(* Logix 5000 project; controller VET 1756-L62 rev 19.52; software revision 19.01; part 6 of 27 *)

        [445].S.BITS2.27   // 9-CON-707 Cmd. Open
        [445].S.BITS2.30   // 9-CON-707 OUT CLOSE
        [445].S.BITS2.31   // 9-CON-707 OUT OPEN
        [447].S.BITS2.31   // 9-CON-709 OUT OPEN
        [450].S.BITS2.31   // 110-VEN-001/2 OUT MARCHA
        [451].S.BITS2.31   // 9-CON-713 OUT OPEN
        [462].S.BITS2.31   // 110-ENF-002/2-4 OUT MARCHA
        [464].S.BITS2.31   // 110-ENF-002/2-1 OUT MARCHA
        [465].S.BITS1.1   // 9-CON-727 Falla Resumen
        [465].S.BITS1.2   // 9-CON-727 Conf Pos Abrir
        [465].S.BITS1.4   // 9-CON-727 Conf Pos Cerrar
        [465].S.BITS1.29   // 9-CON-727 Falla Abrir
        [465].S.BITS1.30   // 9-CON-727 Falla Cerrar
        [465].S.BITS2.20   // 9-CON-727 Reset Falla
        [465].S.BITS2.27   // 9-CON-727 Cmd. Open
        [465].S.BITS2.30   // 9-CON-727 OUT CLOSE
        [465].S.BITS2.31   // 9-CON-727 OUT OPEN
        [467].S.BITS2.31   // 9-CON-729 OUT OPEN
        [471].S.BITS2.31   // 110-ENF-002/2-5 OUT MARCHA
        [474].S.BITS2.31   // 110-TOR-002/2 OUT MARCHA
        [475].S.BITS2.31   // 110-TOR-003/2 OUT MARCHA
        [476].S.BITS2.31   // 110-ELV-002/2 OUT MARCHA
        [478].S.BITS2.31   // 110-TOR-004/2 OUT MARCHA
        [495].S.BITS2.31   // 110-CAN-010/3 OUT MARCHA
        [500].S.BITS2.31   // 110-TOR-001/3 OUT MARCHA
        [502].S.BITS2.31   // 110-ACD-001/3 OUT MARCHA
        [504].S.BITS2.31   // 110-DES-001/3 OUT MARCHA
        [505].S.BITS2.31   // 110-CAE-001/3 OUT MARCHA
        [511].S.BITS2.31   // 110-ESC-001/3 OUT MARCHA
        [512].S.BITS2.31   // 110-ENF-001/3-4 OUT MARCHA
        [514].S.BITS2.31   // 110-ENF-001/3-1 OUT MARCHA
        [515].S.BITS1.1   // 110-ENF-001/3-2 Falla Resumen
        [515].S.BITS1.2   // 110-ENF-001/3-2 Conf Pos Abrir
        [515].S.BITS1.4   // 110-ENF-001/3-2 Conf Pos Cerrar
        [515].S.BITS1.29   // 110-ENF-001/3-2 Falla Abrir
        [515].S.BITS1.30   // 110-ENF-001/3-2 Falla Cerrar
        [515].S.BITS2.20   // 110-ENF-001/3-2 Reset Falla
        [515].S.BITS2.27   // 110-ENF-001/3-2 Cmd. Open
        [515].S.BITS2.30   // 110-ENF-001/3-2 OUT CLOSE
        [515].S.BITS2.31   // 110-ENF-001/3-2 OUT OPEN
        [517].S.BITS2.31   // 110-ESC-003/3 OUT MARCHA
        [519].S.BITS2.31   // 110-VAL-001/3-1 OUT MARCHA
        [520].S.BITS2.31   // 110-VEN-001/3 OUT MARCHA
        [521].S.BITS2.31   // 110-ENF-001/3-5 OUT MARCHA
        [523].S.BITS2.31   // 110-QUE-001-1 OUT MARCHA
        [524].S.BITS2.31   // 110-QUE-001-2 OUT MARCHA
        [531].S.BITS2.31   // 110-ESC-002/3 OUT MARCHA
        [532].S.BITS2.31   // 110-ENF-002/3-4 OUT MARCHA
        [534].S.BITS2.31   // 110-ENF-002/3-1 OUT MARCHA
        [535].S.BITS1.1   // 110-ENF-002/3-2 Falla Resumen
        [535].S.BITS1.2   // 110-ENF-002/3-2 Conf Pos Abrir
        [535].S.BITS1.4   // 110-ENF-002/3-2 Conf Pos Cerrar
        [535].S.BITS1.29   // 110-ENF-002/3-2 Falla Abrir
        [535].S.BITS1.30   // 110-ENF-002/3-2 Falla Cerrar
        [535].S.BITS2.20   // 110-ENF-002/3-2 Reset Falla
        [535].S.BITS2.27   // 110-ENF-002/3-2 Cmd. Open
        [535].S.BITS2.30   // 110-ENF-002/3-2 OUT CLOSE
        [535].S.BITS2.31   // 110-ENF-002/3-2 OUT OPEN
        [537].S.BITS2.31   // 110-ESC-004/3 OUT MARCHA
        [539].S.BITS2.31   // 110-VEN-002/3-1 OUT MARCHA
        [540].S.BITS2.31   // 110-VEN-002/3 OUT MARCHA
        [541].S.BITS2.31   // 110-ENF-002/3-5 OUT MARCHA
        [544].S.BITS2.31   // 110-TOR-002/3 OUT MARCHA
        [545].S.BITS2.31   // 110-TOR-003/3 OUT MARCHA
        [546].S.BITS2.31   // 110-ELV-002/3 OUT MARCHA
        [548].S.BITS2.31   // 110-TOR-004/3 OUT MARCHA
        [551].S.BITS2.31   // 110-TDC-003/1 OUT MARCHA
        [555].S.BITS2.31   // 120-TDC-001/1 OUT MARCHA
        [561].S.BITS2.31   // 110-TDC-003/2 OUT MARCHA
        [562].S.BITS2.31   // 110-TDC-004/2 OUT MARCHA
        [564].S.BITS2.31   // 110-ELV-001/2 OUT MARCHA
        [565].S.BITS2.31   // 120-TDC-001/2 OUT MARCHA
        [571].S.BITS2.31   // 110-TDC-003/3 OUT MARCHA
        [572].S.BITS2.31   // 110-TDC-004/3 OUT MARCHA
        [573].S.BITS2.31   // 110-TDC-005/3 OUT MARCHA
        [574].S.BITS2.31   // 110-ELV-001/3 OUT MARCHA
        [575].S.BITS2.31   // 120-TDC-001/3 OUT MARCHA
        [349].S.BITS1.7   // 110-LRT-001 Puerta
        [383].S.BITS1.14   // Switch de Incendio
        [383].S.BITS1.3   // Alineamiento plataforma
        [383].S.BITS1.11   // Puerta Abierta
        [691].S.BITS1.2   // 100-DOS-100-M13 Conf. Marcha
        [693].S.BITS1.2   // 100-DOS-100-M14 Conf. Marcha
        [1].S.BITS1.4   // 7-LMG-1001 Cmd. Automatico
        [1].S.BITS1.26   // 7-LMG-1001 FLL
        [1].S.BITS1.27   // 7-LMG-1001 FV0
        [1].S.BITS1.28   // 7-LMG-1001 FATO
        [1].S.BITS1.30   // 7-LMG-1001 Falla Partida
        [1].S.BITS2.27   // 7-LMG-1001 Cmd. Marcha
        [1].S.BITS2.20   // 7-LMG-1001 Reset Falla
        [1].S.BITS2.23   // 7-LMG-1001 Test
        [1].S.BITS2.30   // 7-LMG-1001 OUT MARCHA
        [2].S.BITS1.0   // 7-ELV-1002 Enable
        [2].S.BITS1.1   // 7-ELV-1002 Falla Resumen
        [2].S.BITS1.2   // 7-ELV-1002 Conf. Marcha
        [2].S.BITS1.4   // 7-ELV-1002 Cmd. Automatico
        [2].S.BITS1.26   // 7-ELV-1002 FLL
        [2].S.BITS1.27   // 7-ELV-1002 FV0
        [2].S.BITS1.28   // 7-ELV-1002 FATO
        [2].S.BITS1.30   // 7-ELV-1002 Falla Partida
        [2].S.BITS2.27   // 7-ELV-1002 Cmd. Marcha
        [2].S.BITS2.20   // 7-ELV-1002 Reset Falla
        [2].S.BITS2.23   // 7-ELV-1002 Test
        [2].S.BITS2.30   // 7-ELV-1002 OUT MARCHA
        [3].S.BITS1.0   // 7-BIF-1003 Enable
        [3].S.BITS1.1   // 7-BIF-1003 Falla Resumen
        [3].S.BITS1.2   // 7-BIF-1003 Conf. Pos. Izquierda
        [3].S.BITS1.4   // 7-BIF-1003 Conf. Pos. Derecha
        [3].S.BITS1.29   // 7-BIF-1003 Falla Pos. Izquierda
        [3].S.BITS1.30   // 7-BIF-1003 Falla Pos. Derecha
        [3].S.BITS2.20   // 7-BIF-1003 Reset Falla
        [3].S.BITS2.23   // 7-BIF-1003 Test
        [3].S.BITS2.26   // 7-BIF-1003 Cmd. Pos . Izquierda
        [3].S.BITS2.27   // 7-BIF-1003 Cmd. Pos. Derecha
        [3].S.BITS2.30   // 7-BIF-1003 Out Izquierda
        [3].S.BITS2.31   // 7-BIF-1003 Out Derecha
        [5].S.BITS1.26   // 7-RED-1005 FLL
        [5].S.BITS1.27   // 7-RED-1005 FV0
        [5].S.BITS1.28   // 7-RED-1005 FATO
        [5].S.BITS1.30   // 7-RED-1005 Falla Partida
        [5].S.BITS2.27   // 7-RED-1005 Cmd. Marcha
        [5].S.BITS2.30   // 7-RED-1005 OUT MARCHA
        [6].S.BITS2.31   // 7-COM-1006 OUT OPEN
        [8].S.BITS2.31   // 7-COM-1008 OUT OPEN
        [10].S.BITS1.0   // 7-RED-1010 Enable
        [10].S.BITS1.1   // 7-RED-1010 Falla Resumen
        [10].S.BITS1.2   // 7-RED-1010 Conf. Marcha
        [10].S.BITS1.4   // 7-RED-1010 Cmd. Automatico
        [10].S.BITS1.26   // 7-RED-1010 FLL
        [10].S.BITS1.27   // 7-RED-1010 FV0
        [10].S.BITS1.28   // 7-RED-1010 FATO
        [10].S.BITS1.30   // 7-RED-1010 Falla Partida
        [10].S.BITS2.27   // 7-RED-1010 Cmd. Marcha
        [10].S.BITS2.20   // 7-RED-1010 Reset Falla
        [10].S.BITS2.23   // 7-RED-1010 Test
        [10].S.BITS2.30   // 7-RED-1010 OUT MARCHA
        [11].S.BITS1.0   // 7-CON-1011 Enable
        [11].S.BITS1.1   // 7-CON-1011 Falla Resumen
        [11].S.BITS1.2   // 7-CON-1011 Conf Pos Abrir
        [11].S.BITS1.4   // 7-CON-1011 Conf Pos Cerrar
        [11].S.BITS1.29   // 7-CON-1011 Falla Abrir
        [11].S.BITS1.30   // 7-CON-1011 Falla Cerrar
        [11].S.BITS2.20   // 7-CON-1011 Reset Falla
        [11].S.BITS2.23   // 7-CON-1011 Test
        [11].S.BITS2.27   // 7-CON-1011 Cmd. Open
        [11].S.BITS2.30   // 7-CON-1011 OUT CLOSE
        [11].S.BITS2.31   // 7-CON-1011 OUT OPEN
        [12].S.BITS1.0   // 7-CON-1012 Enable
        [12].S.BITS1.1   // 7-CON-1012 Falla Resumen
        [12].S.BITS1.2   // 7-CON-1012 Conf Pos Abrir
        [12].S.BITS1.4   // 7-CON-1012 Conf Pos Cerrar
        [12].S.BITS1.29   // 7-CON-1012 Falla Abrir
        [12].S.BITS1.30   // 7-CON-1012 Falla Cerrar
        [12].S.BITS2.20   // 7-CON-1012 Reset Falla
        [12].S.BITS2.23   // 7-CON-1012 Test
        [12].S.BITS2.27   // 7-CON-1012 Cmd. Open
        [12].S.BITS2.30   // 7-CON-1012 OUT CLOSE
        [12].S.BITS2.31   // 7-CON-1012 OUT OPEN
        [13].S.BITS1.2   // 7-CON-1013 Conf Pos Abrir
        [15].S.BITS1.0   // 7-BIF-1023a Enable
        [15].S.BITS1.1   // 7-BIF-1023a Falla Resumen
        [15].S.BITS1.2   // 7-BIF-1023a Conf. Pos. Izquierda
        [15].S.BITS1.4   // 7-BIF-1023a Conf. Pos. Derecha
        [15].S.BITS1.29   // 7-BIF-1023a Falla Pos. Izquierda
        [15].S.BITS1.30   // 7-BIF-1023a Falla Pos. Derecha
        [15].S.BITS2.20   // 7-BIF-1023a Reset Falla
        [15].S.BITS2.23   // 7-BIF-1023a Test
        [15].S.BITS2.26   // 7-BIF-1023a Cmd. Pos . Izquierda
        [15].S.BITS2.27   // 7-BIF-1023a Cmd. Pos. Derecha
        [15].S.BITS2.30   // 7-BIF-1023a Out Izquierda
        [15].S.BITS2.31   // 7-BIF-1023a Out Derecha
        [16].S.BITS1.26   // 7-LMG-1016 FLL
        [16].S.BITS1.27   // 7-LMG-1016 FV0
        [16].S.BITS1.28   // 7-LMG-1016 FATO
        [16].S.BITS1.30   // 7-LMG-1016 Falla Partida
        [16].S.BITS2.27   // 7-LMG-1016 Cmd. Marcha
        [16].S.BITS2.30   // 7-LMG-1016 OUT MARCHA
        [17].S.BITS1.26   // 7-ELV-1017 FLL
        [17].S.BITS1.27   // 7-ELV-1017 FV0
        [17].S.BITS1.28   // 7-ELV-1017 FATO
        [17].S.BITS1.30   // 7-ELV-1017 Falla Partida
        [17].S.BITS2.27   // 7-ELV-1017 Cmd. Marcha
        [17].S.BITS2.30   // 7-ELV-1017 OUT MARCHA
        [18].S.BITS1.2   // 7-BIF-1018 Conf. Pos. Izquierda
        [18].S.BITS1.4   // 7-BIF-1018 Conf. Pos. Derecha
        [18].S.BITS1.29   // 7-BIF-1018 Falla Pos. Izquierda
        [18].S.BITS1.30   // 7-BIF-1018 Falla Pos. Derecha
        [18].S.BITS2.26   // 7-BIF-1018 Cmd. Pos . Izquierda
        [18].S.BITS2.27   // 7-BIF-1018 Cmd. Pos. Derecha
        [18].S.BITS2.30   // 7-BIF-1018 Out Izquierda
        [18].S.BITS2.31   // 7-BIF-1018 Out Derecha
        [19].S.BITS1.26   // 7-RED-1019 FLL
        [19].S.BITS1.27   // 7-RED-1019 FV0
        [19].S.BITS1.28   // 7-RED-1019 FATO
        [19].S.BITS1.30   // 7-RED-1019 Falla Partida
        [19].S.BITS2.27   // 7-RED-1019 Cmd. Marcha
        [19].S.BITS2.30   // 7-RED-1019 OUT MARCHA
        [20].S.BITS1.26   // 7-RED-1020 FLL
        [20].S.BITS1.27   // 7-RED-1020 FV0
        [20].S.BITS1.28   // 7-RED-1020 FATO
        [20].S.BITS1.30   // 7-RED-1020 Falla Partida
        [20].S.BITS2.27   // 7-RED-1020 Cmd. Marcha
        [20].S.BITS2.30   // 7-RED-1020 OUT MARCHA
        [24].S.BITS1.26   // 7-RED-1024 FLL
        [24].S.BITS1.27   // 7-RED-1024 FV0
        [24].S.BITS1.28   // 7-RED-1024 FATO
        [24].S.BITS1.30   // 7-RED-1024 Falla Partida
        [24].S.BITS2.27   // 7-RED-1024 Cmd. Marcha
        [24].S.BITS2.30   // 7-RED-1024 OUT MARCHA
        [26].S.BITS1.2   // 7-CON-1026 Conf Pos Abrir
        [26].S.BITS1.29   // 7-CON-1026 Falla Abrir
        [27].S.BITS1.2   // 7-BIF-1027 Conf. Pos. Izquierda
        [27].S.BITS1.4   // 7-BIF-1027 Conf. Pos. Derecha
        [27].S.BITS1.29   // 7-BIF-1027 Falla Pos. Izquierda
        [27].S.BITS1.30   // 7-BIF-1027 Falla Pos. Derecha
        [27].S.BITS2.26   // 7-BIF-1027 Cmd. Pos . Izquierda
        [27].S.BITS2.27   // 7-BIF-1027 Cmd. Pos. Derecha
        [27].S.BITS2.30   // 7-BIF-1027 Out Izquierda
        [27].S.BITS2.31   // 7-BIF-1027 Out Derecha
        [30].S.BITS1.0   // 7-ELV-1051 Enable
        [30].S.BITS1.1   // 7-ELV-1051 Falla Resumen
        [30].S.BITS1.2   // 7-ELV-1051 Conf. Marcha
        [30].S.BITS1.4   // 7-ELV-1051 Cmd. Automatico
        [30].S.BITS1.26   // 7-ELV-1051 FLL
        [30].S.BITS1.27   // 7-ELV-1051 FV0
        [30].S.BITS1.28   // 7-ELV-1051 FATO
        [30].S.BITS1.30   // 7-ELV-1051 Falla Partida
        [30].S.BITS2.27   // 7-ELV-1051 Cmd. Marcha
        [30].S.BITS2.20   // 7-ELV-1051 Reset Falla
        [30].S.BITS2.23   // 7-ELV-1051 Test
        [30].S.BITS2.30   // 7-ELV-1051 OUT MARCHA
        [32].S.BITS1.2   // 7-RED-1053 Conf. Marcha
        [32].S.BITS1.26   // 7-RED-1053 FLL
        [32].S.BITS1.27   // 7-RED-1053 FV0
        [32].S.BITS1.28   // 7-RED-1053 FATO
        [32].S.BITS1.30   // 7-RED-1053 Falla Partida
        [32].S.BITS2.27   // 7-RED-1053 Cmd. Marcha
        [32].S.BITS2.30   // 7-RED-1053 OUT MARCHA
        [33].S.BITS1.2   // 7-CON-1054 Conf Pos Abrir
        [33].S.BITS1.29   // 7-CON-1054 Falla Abrir
        [33].S.BITS2.31   // 7-CON-1054 OUT OPEN
        [34].S.BITS1.2   // 7-BIF-1055 Conf. Pos. Izquierda
        [34].S.BITS1.4   // 7-BIF-1055 Conf. Pos. Derecha
        [34].S.BITS1.29   // 7-BIF-1055 Falla Pos. Izquierda
        [34].S.BITS1.30   // 7-BIF-1055 Falla Pos. Derecha
        [34].S.BITS2.26   // 7-BIF-1055 Cmd. Pos . Izquierda
        [34].S.BITS2.27   // 7-BIF-1055 Cmd. Pos. Derecha
        [34].S.BITS2.30   // 7-BIF-1055 Out Izquierda
        [34].S.BITS2.31   // 7-BIF-1055 Out Derecha
        [38].S.BITS1.8   // 7-BIN-1062 LL
        [38].S.BITS1.9   // 7-BIN-1062 LM
        [38].S.BITS1.10   // 7-BIN-1062 LH
        [41].S.BITS1.30   // 7-MMA-1065 Falla Partida
        [41].S.BITS2.27   // 7-MMA-1065 Cmd. Marcha
        [41].S.BITS2.30   // 7-MMA-1065 OUT MARCHA
        [42].S.BITS1.26   // 7-FLT-1066 FLL
        [42].S.BITS1.27   // 7-FLT-1066 FV0
        [42].S.BITS1.28   // 7-FLT-1066 FATO
        [42].S.BITS1.30   // 7-FLT-1066 Falla Partida
        [42].S.BITS2.27   // 7-FLT-1066 Cmd. Marcha
        [42].S.BITS2.30   // 7-FLT-1066 OUT MARCHA
        [44].S.BITS1.8   // 7-TV-107X LL
        [47].S.BITS1.2   // 7-ELV-1070 Conf. Marcha
        [48].S.BITS1.0   // 7-RED-1071 Enable
        [48].S.BITS1.1   // 7-RED-1071 Falla Resumen
        [48].S.BITS1.2   // 7-RED-1071 Conf. Marcha
        [48].S.BITS1.4   // 7-RED-1071 Cmd. Automatico
        [48].S.BITS1.30   // 7-RED-1071 Falla Partida
        [48].S.BITS2.27   // 7-RED-1071 Cmd. Marcha
        [48].S.BITS2.20   // 7-RED-1071 Reset Falla
        [48].S.BITS2.23   // 7-RED-1071 Test
        [48].S.BITS2.30   // 7-RED-1071 OUT MARCHA
        [49].S.BITS1.2   // 7-CON-1072 Conf Pos Abrir
        [49].S.BITS1.29   // 7-CON-1072 Falla Abrir
        [50].S.BITS1.2   // 7-CON-1073 Conf Pos Abrir
        [50].S.BITS1.29   // 7-CON-1073 Falla Abrir
        [51].S.BITS2.30   // 7-CON-1074 OUT CLOSE
        [51].S.BITS2.31   // 7-CON-1074 OUT OPEN
        [53].S.BITS1.30   // 7-RED-1076 Falla Partida
        [53].S.BITS2.27   // 7-RED-1076 Cmd. Marcha
        [53].S.BITS2.30   // 7-RED-1076 OUT MARCHA
        [54].S.BITS1.2   // 7-CON-1077 Conf Pos Abrir
        [54].S.BITS1.29   // 7-CON-1077 Falla Abrir
        [55].S.BITS1.30   // 7-RED-1078 Falla Partida
        [55].S.BITS2.27   // 7-RED-1078 Cmd. Marcha
        [55].S.BITS2.30   // 7-RED-1078 OUT MARCHA
        [56].S.BITS1.2   // 7-CON-1079 Conf Pos Abrir
        [57].S.BITS1.2   // 7-CON-1080 Conf Pos Abrir
        [57].S.BITS1.29   // 7-CON-1080 Falla Abrir
        [61].S.BITS1.0   // 7-MRO-1083a Enable
        [61].S.BITS1.1   // 7-MRO-1083a Falla Resumen
        [61].S.BITS1.4   // 7-MRO-1083a Cmd. Automatico
        [61].S.BITS1.26   // 7-MRO-1083a FLL
        [61].S.BITS1.27   // 7-MRO-1083a FV0
        [61].S.BITS1.28   // 7-MRO-1083a FATO
        [61].S.BITS1.30   // 7-MRO-1083a Falla Partida
        [61].S.BITS2.27   // 7-MRO-1083a Cmd. Marcha
        [61].S.BITS2.20   // 7-MRO-1083a Reset Falla
        [61].S.BITS2.23   // 7-MRO-1083a Test
        [61].S.BITS2.30   // 7-MRO-1083a OUT MARCHA
        [62].S.BITS1.0   // 7-MRO-1083b Enable
        [62].S.BITS1.1   // 7-MRO-1083b Falla Resumen
        [62].S.BITS1.2   // 7-MRO-1083b Conf. Marcha
        [62].S.BITS1.4   // 7-MRO-1083b Cmd. Automatico
        [62].S.BITS1.26   // 7-MRO-1083b FLL
        [62].S.BITS1.27   // 7-MRO-1083b FV0
        [62].S.BITS1.28   // 7-MRO-1083b FATO
        [62].S.BITS1.30   // 7-MRO-1083b Falla Partida
        [62].S.BITS2.27   // 7-MRO-1083b Cmd. Marcha
        [62].S.BITS2.20   // 7-MRO-1083b Reset Falla
        [62].S.BITS2.23   // 7-MRO-1083b Test
        [62].S.BITS2.30   // 7-MRO-1083b OUT MARCHA
        [67].S.BITS1.0   // 7-MRO-1086a Enable
        [67].S.BITS1.1   // 7-MRO-1086a Falla Resumen
        [67].S.BITS1.2   // 7-MRO-1086a Conf. Marcha
        [67].S.BITS1.4   // 7-MRO-1086a Cmd. Automatico
        [67].S.BITS1.26   // 7-MRO-1086a FLL
        [67].S.BITS1.27   // 7-MRO-1086a FV0
        [67].S.BITS1.28   // 7-MRO-1086a FATO
        [67].S.BITS1.30   // 7-MRO-1086a Falla Partida
        [67].S.BITS2.27   // 7-MRO-1086a Cmd. Marcha
        [67].S.BITS2.20   // 7-MRO-1086a Reset Falla
        [67].S.BITS2.23   // 7-MRO-1086a Test
        [67].S.BITS2.30   // 7-MRO-1086a OUT MARCHA
        [68].S.BITS1.0   // 7-MRO-1086b Enable
        [68].S.BITS1.1   // 7-MRO-1086b Falla Resumen
        [68].S.BITS1.2   // 7-MRO-1086b Conf. Marcha
        [68].S.BITS1.4   // 7-MRO-1086b Cmd. Automatico
        [68].S.BITS1.26   // 7-MRO-1086b FLL
        [68].S.BITS1.27   // 7-MRO-1086b FV0
        [68].S.BITS1.28   // 7-MRO-1086b FATO
        [68].S.BITS1.30   // 7-MRO-1086b Falla Partida
        [68].S.BITS2.27   // 7-MRO-1086b Cmd. Marcha
        [68].S.BITS2.20   // 7-MRO-1086b Reset Falla
        [68].S.BITS2.23   // 7-MRO-1086b Test
        [68].S.BITS2.30   // 7-MRO-1086b OUT MARCHA
        [69].S.BITS1.0   // 7-MRO-1086c Enable
        [69].S.BITS1.1   // 7-MRO-1086c Falla Resumen
        [69].S.BITS1.2   // 7-MRO-1086c Conf. Marcha
        [69].S.BITS1.4   // 7-MRO-1086c Cmd. Automatico
        [69].S.BITS1.26   // 7-MRO-1086c FLL
        [69].S.BITS1.27   // 7-MRO-1086c FV0
        [69].S.BITS1.28   // 7-MRO-1086c FATO
        [69].S.BITS1.30   // 7-MRO-1086c Falla Partida
        [69].S.BITS2.27   // 7-MRO-1086c Cmd. Marcha
        [69].S.BITS2.20   // 7-MRO-1086c Reset Falla
        [69].S.BITS2.23   // 7-MRO-1086c Test
        [69].S.BITS2.30   // 7-MRO-1086c OUT MARCHA
        [70].S.BITS1.0   // 7-MRO-1086d Enable
        [70].S.BITS1.1   // 7-MRO-1086d Falla Resumen
        [70].S.BITS1.2   // 7-MRO-1086d Conf. Marcha
        [70].S.BITS1.4   // 7-MRO-1086d Cmd. Automatico
        [70].S.BITS1.26   // 7-MRO-1086d FLL
        [70].S.BITS1.27   // 7-MRO-1086d FV0
        [70].S.BITS1.28   // 7-MRO-1086d FATO
        [70].S.BITS1.30   // 7-MRO-1086d Falla Partida
        [70].S.BITS2.27   // 7-MRO-1086d Cmd. Marcha
        [70].S.BITS2.20   // 7-MRO-1086d Reset Falla
        [70].S.BITS2.23   // 7-MRO-1086d Test
        [70].S.BITS2.30   // 7-MRO-1086d OUT MARCHA
        [71].S.BITS1.9   // 7-BIN-1087 LM
        [76].S.BITS1.0   // 7-MRO-1089d Enable
        [76].S.BITS1.1   // 7-MRO-1089d Falla Resumen
        [76].S.BITS1.2   // 7-MRO-1089d Conf. Marcha
        [76].S.BITS1.4   // 7-MRO-1089d Cmd. Automatico
        [76].S.BITS1.26   // 7-MRO-1089d FLL
        [76].S.BITS1.27   // 7-MRO-1089d FV0
        [76].S.BITS1.28   // 7-MRO-1089d FATO
        [76].S.BITS1.30   // 7-MRO-1089d Falla Partida
        [76].S.BITS2.27   // 7-MRO-1089d Cmd. Marcha
        [76].S.BITS2.20   // 7-MRO-1089d Reset Falla
        [76].S.BITS2.23   // 7-MRO-1089d Test
        [76].S.BITS2.30   // 7-MRO-1089d OUT MARCHA
        [77].S.BITS1.26   // 7-RED-1090 FLL
        [77].S.BITS1.27   // 7-RED-1090 FV0
        [77].S.BITS1.28   // 7-RED-1090 FATO
        [79].S.BITS1.26   // 7-ELV-1092 FLL
        [79].S.BITS1.27   // 7-ELV-1092 FV0
        [79].S.BITS1.28   // 7-ELV-1092 FATO
        [79].S.BITS1.30   // 7-ELV-1092 Falla Partida
        [79].S.BITS2.27   // 7-ELV-1092 Cmd. Marcha
        [79].S.BITS2.30   // 7-ELV-1092 OUT MARCHA
        [80].S.BITS1.2   // 7-RED-1093 Conf. Marcha
        [80].S.BITS1.26   // 7-RED-1093 FLL
        [80].S.BITS1.27   // 7-RED-1093 FV0
        [80].S.BITS1.28   // 7-RED-1093 FATO
        [80].S.BITS1.30   // 7-RED-1093 Falla Partida
        [80].S.BITS2.27   // 7-RED-1093 Cmd. Marcha
        [80].S.BITS2.30   // 7-RED-1093 OUT MARCHA
        [82].S.BITS1.2   // 7-CON-1095 Conf Pos Abrir
        [82].S.BITS1.29   // 7-CON-1095 Falla Abrir
        [83].S.BITS1.29   // 7-CON-1096 Falla Abrir
        [86].S.BITS1.26   // tcs-28_M FLL
        [86].S.BITS1.27   // tcs-28_M FV0
        [86].S.BITS1.28   // tcs-28_M FATO
        [89].S.BITS1.8   // 7-TOL-010 LL
        [90].S.BITS1.8   // 7-TOL-011 LL
        [90].S.BITS1.9   // 7-TOL-011 LM
        [90].S.BITS1.10   // 7-TOL-011 LH
        [91].S.BITS1.8   // 7-TOL-012 LL
        [91].S.BITS1.9   // 7-TOL-012 LM
        [91].S.BITS1.10   // 7-TOL-012 LH
        [95].S.BITS1.9   // 7-RED-770 LM
        [97].S.BITS1.8   // 7-TOL-799 LL
        [110].S.BITS1.0   // 7-ROS-1109 Enable
        [110].S.BITS1.1   // 7-ROS-1109 Falla Resumen
        [110].S.BITS1.4   // 7-ROS-1109 Cmd. Automatico
        [110].S.BITS1.26   // 7-ROS-1109 FLL
        [110].S.BITS1.27   // 7-ROS-1109 FV0
        [110].S.BITS1.28   // 7-ROS-1109 FATO
        [110].S.BITS1.30   // 7-ROS-1109 Falla Partida
        [110].S.BITS2.27   // 7-ROS-1109 Cmd. Marcha
        [110].S.BITS2.20   // 7-ROS-1109 Reset Falla
        [110].S.BITS2.23   // 7-ROS-1109 Test
        [110].S.BITS2.30   // 7-ROS-1109 OUT MARCHA
        [111].S.BITS1.8   // 7-BIN-1110 LL
        [111].S.BITS1.9   // 7-BIN-1110 LM
        [111].S.BITS1.10   // 7-BIN-1110 LH
        [114].S.BITS1.0   // 7-ROS-1113 Enable
        [114].S.BITS1.1   // 7-ROS-1113 Falla Resumen
        [114].S.BITS1.4   // 7-ROS-1113 Cmd. Automatico
        [114].S.BITS1.26   // 7-ROS-1113 FLL
        [114].S.BITS1.27   // 7-ROS-1113 FV0
        [114].S.BITS1.28   // 7-ROS-1113 FATO
        [114].S.BITS1.30   // 7-ROS-1113 Falla Partida
        [114].S.BITS2.27   // 7-ROS-1113 Cmd. Marcha
        [114].S.BITS2.20   // 7-ROS-1113 Reset Falla
        [114].S.BITS2.23   // 7-ROS-1113 Test
        [114].S.BITS2.30   // 7-ROS-1113 OUT MARCHA
        [117].S.BITS1.8   // 7-BIN-1116 LL
        [118].S.BITS1.0   // 7-ROS-1117 Enable
        [118].S.BITS1.1   // 7-ROS-1117 Falla Resumen
        [118].S.BITS1.2   // 7-ROS-1117 Conf. Marcha
        [118].S.BITS1.4   // 7-ROS-1117 Cmd. Automatico
        [118].S.BITS1.26   // 7-ROS-1117 FLL
        [118].S.BITS1.27   // 7-ROS-1117 FV0
        [118].S.BITS1.28   // 7-ROS-1117 FATO
        [118].S.BITS1.30   // 7-ROS-1117 Falla Partida
        [118].S.BITS2.27   // 7-ROS-1117 Cmd. Marcha
        [118].S.BITS2.20   // 7-ROS-1117 Reset Falla
        [118].S.BITS2.23   // 7-ROS-1117 Test
        [118].S.BITS2.30   // 7-ROS-1117 OUT MARCHA
        [119].S.BITS1.8   // 7-BIN-1118 LL
        [119].S.BITS1.9   // 7-BIN-1118 LM
        [119].S.BITS1.10   // 7-BIN-1118 LH
        [120].S.BITS1.0   // 7-ROS-1119 Enable
        [120].S.BITS1.1   // 7-ROS-1119 Falla Resumen
        [120].S.BITS1.4   // 7-ROS-1119 Cmd. Automatico
        [120].S.BITS1.26   // 7-ROS-1119 FLL
        [120].S.BITS1.27   // 7-ROS-1119 FV0
        [120].S.BITS1.28   // 7-ROS-1119 FATO
        [120].S.BITS1.30   // 7-ROS-1119 Falla Partida
        [120].S.BITS2.27   // 7-ROS-1119 Cmd. Marcha
        [120].S.BITS2.20   // 7-ROS-1119 Reset Falla
        [120].S.BITS2.23   // 7-ROS-1119 Test
        [120].S.BITS2.30   // 7-ROS-1119 OUT MARCHA
        [121].S.BITS1.9   // 7-BIN-1120 LM
        [123].S.BITS1.8   // 7-BIN-1122 LL
        [124].S.BITS1.26   // 7-ROS-1123 FLL
        [124].S.BITS1.27   // 7-ROS-1123 FV0
        [124].S.BITS1.28   // 7-ROS-1123 FATO
        [124].S.BITS2.27   // 7-ROS-1123 Cmd. Marcha
        [125].S.BITS1.9   // 7-BIN-1124 LM
        [128].S.BITS1.26   // 7-ROS-1127 FLL
        [128].S.BITS1.27   // 7-ROS-1127 FV0
        [128].S.BITS1.28   // 7-ROS-1127 FATO
        [128].S.BITS2.27   // 7-ROS-1127 Cmd. Marcha
        [129].S.BITS1.9   // 7-BIN-1128 LM
        [133].S.BITS1.8   // 7-TOL-1134 LL
        [140].S.BITS1.0   // 7-VEN-1154 Enable
        [140].S.BITS1.1   // 7-VEN-1154 Falla Resumen
        [140].S.BITS1.2   // 7-VEN-1154 Conf. Marcha
        [140].S.BITS1.4   // 7-VEN-1154 Cmd. Automatico
        [140].S.BITS1.26   // 7-VEN-1154 FLL
        [140].S.BITS1.27   // 7-VEN-1154 FV0
        [140].S.BITS1.28   // 7-VEN-1154 FATO
        [140].S.BITS1.30   // 7-VEN-1154 Falla Partida
        [140].S.BITS2.27   // 7-VEN-1154 Cmd. Marcha
        [140].S.BITS2.20   // 7-VEN-1154 Reset Falla
        [140].S.BITS2.23   // 7-VEN-1154 Test
        [140].S.BITS2.30   // 7-VEN-1154 OUT MARCHA
        [143].S.BITS2.27   // 7-BBA-1142 Cmd. Marcha
        [144].S.BITS1.26   // 7-RED-1143 FLL
        [144].S.BITS1.27   // 7-RED-1143 FV0
        [144].S.BITS1.28   // 7-RED-1143 FATO
        [144].S.BITS2.27   // 7-RED-1143 Cmd. Marcha
        [145].S.BITS1.2   // 7-BIF-1144 Conf. Pos. Izquierda
        [145].S.BITS1.4   // 7-BIF-1144 Conf. Pos. Derecha
        [145].S.BITS1.29   // 7-BIF-1144 Falla Pos. Izquierda
        [145].S.BITS1.30   // 7-BIF-1144 Falla Pos. Derecha
        [145].S.BITS2.26   // 7-BIF-1144 Cmd. Pos . Izquierda
        [145].S.BITS2.27   // 7-BIF-1144 Cmd. Pos. Derecha
        [145].S.BITS2.30   // 7-BIF-1144 Out Izquierda
        [145].S.BITS2.31   // 7-BIF-1144 Out Derecha
        [149].S.BITS1.2   // 7-CON-1148 Conf Pos Abrir
        [149].S.BITS1.29   // 7-CON-1148 Falla Abrir
        [149].S.BITS2.31   // 7-CON-1148 OUT OPEN
        [150].S.BITS1.0   // 7-RED-1150 Enable
        [150].S.BITS1.1   // 7-RED-1150 Falla Resumen
        [150].S.BITS1.2   // 7-RED-1150 Conf. Marcha
        [150].S.BITS1.4   // 7-RED-1150 Cmd. Automatico
        [150].S.BITS1.26   // 7-RED-1150 FLL
        [150].S.BITS1.27   // 7-RED-1150 FV0
        [150].S.BITS1.28   // 7-RED-1150 FATO
        [150].S.BITS1.30   // 7-RED-1150 Falla Partida
        [150].S.BITS2.27   // 7-RED-1150 Cmd. Marcha
        [150].S.BITS2.20   // 7-RED-1150 Reset Falla
        [150].S.BITS2.23   // 7-RED-1150 Test
        [150].S.BITS2.30   // 7-RED-1150 OUT MARCHA
        [151].S.BITS1.2   // 7-CON-1151 Conf Pos Abrir
        [151].S.BITS1.29   // 7-CON-1151 Falla Abrir
        [151].S.BITS2.31   // 7-CON-1151 OUT OPEN
        [152].S.BITS1.2   // 7-CON-1152 Conf Pos Abrir
        [152].S.BITS1.29   // 7-CON-1152 Falla Abrir
        [154].S.BITS1.26   // 7-ELV-1149 FLL
        [154].S.BITS1.27   // 7-ELV-1149 FV0
        [154].S.BITS1.28   // 7-ELV-1149 FATO
        [154].S.BITS2.27   // 7-ELV-1149 Cmd. Marcha
        [159].S.BITS2.27   // 7-ROS-1158 Cmd. Marcha
        [163].S.BITS2.27   // 7-ROS-1162 Cmd. Marcha
        [174].S.BITS1.8   // 7-DOS-1170-01 LL
        [174].S.BITS1.9   // 7-DOS-1170-01 LM
        [174].S.BITS1.10   // 7-DOS-1170-01 LH
        [175].S.BITS1.0   // 7-DOS-1170-01 Enable
        [175].S.BITS1.1   // 7-DOS-1170-01 Falla Resumen
        [175].S.BITS1.2   // 7-DOS-1170-01 Conf. Marcha
        [175].S.BITS1.4   // 7-DOS-1170-01 Cmd. Automatico
        [175].S.BITS1.26   // 7-DOS-1170-01 FLL
        [175].S.BITS1.27   // 7-DOS-1170-01 FV0
        [175].S.BITS1.28   // 7-DOS-1170-01 FATO
        [175].S.BITS1.30   // 7-DOS-1170-01 Falla Partida
        [175].S.BITS2.27   // 7-DOS-1170-01 Cmd. Marcha
        [175].S.BITS2.20   // 7-DOS-1170-01 Reset Falla
        [175].S.BITS2.23   // 7-DOS-1170-01 Test
        [175].S.BITS2.30   // 7-DOS-1170-01 OUT MARCHA
        [176].S.BITS1.8   // 7-DOS-1170-02 LL
        [176].S.BITS1.9   // 7-DOS-1170-02 LM
        [176].S.BITS1.10   // 7-DOS-1170-02 LH
        [177].S.BITS1.0   // 7-DOS-1170-02 Enable
        [177].S.BITS1.1   // 7-DOS-1170-02 Falla Resumen
        [177].S.BITS1.2   // 7-DOS-1170-02 Conf. Marcha
        [177].S.BITS1.4   // 7-DOS-1170-02 Cmd. Automatico
        [177].S.BITS1.26   // 7-DOS-1170-02 FLL
        [177].S.BITS1.27   // 7-DOS-1170-02 FV0
        [177].S.BITS1.28   // 7-DOS-1170-02 FATO
        [177].S.BITS1.30   // 7-DOS-1170-02 Falla Partida
        [177].S.BITS2.27   // 7-DOS-1170-02 Cmd. Marcha
        [177].S.BITS2.20   // 7-DOS-1170-02 Reset Falla
        [177].S.BITS2.23   // 7-DOS-1170-02 Test
        [177].S.BITS2.30   // 7-DOS-1170-02 OUT MARCHA
        [179].S.BITS1.0   // 7-DOS-1170-03 Enable
        [179].S.BITS1.1   // 7-DOS-1170-03 Falla Resumen
        [179].S.BITS1.2   // 7-DOS-1170-03 Conf. Marcha
        [179].S.BITS1.4   // 7-DOS-1170-03 Cmd. Automatico
        [179].S.BITS1.26   // 7-DOS-1170-03 FLL
        [179].S.BITS1.27   // 7-DOS-1170-03 FV0
        [179].S.BITS1.28   // 7-DOS-1170-03 FATO
        [179].S.BITS1.30   // 7-DOS-1170-03 Falla Partida
        [179].S.BITS2.27   // 7-DOS-1170-03 Cmd. Marcha
        [179].S.BITS2.20   // 7-DOS-1170-03 Reset Falla
        [179].S.BITS2.23   // 7-DOS-1170-03 Test
        [179].S.BITS2.30   // 7-DOS-1170-03 OUT MARCHA
        [180].S.BITS1.8   // 7-DOS-1170-04 LL
        [180].S.BITS1.9   // 7-DOS-1170-04 LM
        [180].S.BITS1.10   // 7-DOS-1170-04 LH
        [181].S.BITS1.0   // 7-DOS-1170-04 Enable
        [181].S.BITS1.1   // 7-DOS-1170-04 Falla Resumen
        [181].S.BITS1.2   // 7-DOS-1170-04 Conf. Marcha
        [181].S.BITS1.4   // 7-DOS-1170-04 Cmd. Automatico
        [181].S.BITS1.26   // 7-DOS-1170-04 FLL
        [181].S.BITS1.27   // 7-DOS-1170-04 FV0
        [181].S.BITS1.28   // 7-DOS-1170-04 FATO
        [181].S.BITS1.30   // 7-DOS-1170-04 Falla Partida
        [181].S.BITS2.27   // 7-DOS-1170-04 Cmd. Marcha
        [181].S.BITS2.20   // 7-DOS-1170-04 Reset Falla
        [181].S.BITS2.23   // 7-DOS-1170-04 Test
        [181].S.BITS2.30   // 7-DOS-1170-04 OUT MARCHA
        [183].S.BITS1.0   // 7-DOS-1170-05 Enable
        [183].S.BITS1.1   // 7-DOS-1170-05 Falla Resumen
        [183].S.BITS1.2   // 7-DOS-1170-05 Conf. Marcha
        [183].S.BITS1.4   // 7-DOS-1170-05 Cmd. Automatico
        [183].S.BITS1.26   // 7-DOS-1170-05 FLL
        [183].S.BITS1.27   // 7-DOS-1170-05 FV0
        [183].S.BITS1.28   // 7-DOS-1170-05 FATO
        [183].S.BITS1.30   // 7-DOS-1170-05 Falla Partida
        [183].S.BITS2.27   // 7-DOS-1170-05 Cmd. Marcha
        [183].S.BITS2.20   // 7-DOS-1170-05 Reset Falla
        [183].S.BITS2.23   // 7-DOS-1170-05 Test
        [183].S.BITS2.30   // 7-DOS-1170-05 OUT MARCHA
        [185].S.BITS1.0   // 7-DOS-1170-06 Enable
        [185].S.BITS1.1   // 7-DOS-1170-06 Falla Resumen
        [185].S.BITS1.2   // 7-DOS-1170-06 Conf. Marcha
        [185].S.BITS1.4   // 7-DOS-1170-06 Cmd. Automatico
        [185].S.BITS1.26   // 7-DOS-1170-06 FLL
        [185].S.BITS1.27   // 7-DOS-1170-06 FV0
        [185].S.BITS1.28   // 7-DOS-1170-06 FATO
        [185].S.BITS1.30   // 7-DOS-1170-06 Falla Partida
        [185].S.BITS2.27   // 7-DOS-1170-06 Cmd. Marcha
        [185].S.BITS2.20   // 7-DOS-1170-06 Reset Falla
        [185].S.BITS2.23   // 7-DOS-1170-06 Test
        [185].S.BITS2.30   // 7-DOS-1170-06 OUT MARCHA
        [186].S.BITS1.8   // 7-DOS-1170-07 LL
        [186].S.BITS1.9   // 7-DOS-1170-07 LM
        [186].S.BITS1.10   // 7-DOS-1170-07 LH
        [187].S.BITS1.0   // 7-DOS-1170-07 Enable
        [187].S.BITS1.1   // 7-DOS-1170-07 Falla Resumen
        [187].S.BITS1.2   // 7-DOS-1170-07 Conf. Marcha
        [187].S.BITS1.4   // 7-DOS-1170-07 Cmd. Automatico
        [187].S.BITS1.26   // 7-DOS-1170-07 FLL
        [187].S.BITS1.27   // 7-DOS-1170-07 FV0
        [187].S.BITS1.28   // 7-DOS-1170-07 FATO
        [187].S.BITS1.30   // 7-DOS-1170-07 Falla Partida
        [187].S.BITS2.27   // 7-DOS-1170-07 Cmd. Marcha
        [187].S.BITS2.20   // 7-DOS-1170-07 Reset Falla
        [187].S.BITS2.23   // 7-DOS-1170-07 Test
        [187].S.BITS2.30   // 7-DOS-1170-07 OUT MARCHA
        [188].S.BITS1.8   // 7-DOS-1170-08 LL
        [188].S.BITS1.9   // 7-DOS-1170-08 LM
        [188].S.BITS1.10   // 7-DOS-1170-08 LH
        [189].S.BITS1.0   // 7-DOS-1170-08 Enable
        [189].S.BITS1.1   // 7-DOS-1170-08 Falla Resumen
        [189].S.BITS1.2   // 7-DOS-1170-08 Conf. Marcha
        [189].S.BITS1.4   // 7-DOS-1170-08 Cmd. Automatico
        [189].S.BITS1.26   // 7-DOS-1170-08 FLL
        [189].S.BITS1.27   // 7-DOS-1170-08 FV0
        [189].S.BITS1.28   // 7-DOS-1170-08 FATO
        [189].S.BITS1.30   // 7-DOS-1170-08 Falla Partida
        [189].S.BITS2.27   // 7-DOS-1170-08 Cmd. Marcha
        [189].S.BITS2.20   // 7-DOS-1170-08 Reset Falla
        [189].S.BITS2.23   // 7-DOS-1170-08 Test
        [189].S.BITS2.30   // 7-DOS-1170-08 OUT MARCHA
        [190].S.BITS1.8   // 7-DOS-1170-09 LL
        [190].S.BITS1.9   // 7-DOS-1170-09 LM
        [190].S.BITS1.10   // 7-DOS-1170-09 LH
        [191].S.BITS1.0   // 7-DOS-1170-09 Enable
        [191].S.BITS1.1   // 7-DOS-1170-09 Falla Resumen
        [191].S.BITS1.2   // 7-DOS-1170-09 Conf. Marcha
        [191].S.BITS1.4   // 7-DOS-1170-09 Cmd. Automatico
        [191].S.BITS1.26   // 7-DOS-1170-09 FLL
        [191].S.BITS1.27   // 7-DOS-1170-09 FV0
        [191].S.BITS1.28   // 7-DOS-1170-09 FATO
        [191].S.BITS1.30   // 7-DOS-1170-09 Falla Partida
        [191].S.BITS2.27   // 7-DOS-1170-09 Cmd. Marcha
        [191].S.BITS2.20   // 7-DOS-1170-09 Reset Falla
        [191].S.BITS2.23   // 7-DOS-1170-09 Test
        [191].S.BITS2.30   // 7-DOS-1170-09 OUT MARCHA
        [192].S.BITS1.8   // 7-DOS-1170-10 LL
        [192].S.BITS1.9   // 7-DOS-1170-10 LM
        [192].S.BITS1.10   // 7-DOS-1170-10 LH
        [193].S.BITS1.0   // 7-DOS-1170-10 Enable
        [193].S.BITS1.1   // 7-DOS-1170-10 Falla Resumen
        [193].S.BITS1.2   // 7-DOS-1170-10 Conf. Marcha
        [193].S.BITS1.4   // 7-DOS-1170-10 Cmd. Automatico
        [193].S.BITS1.26   // 7-DOS-1170-10 FLL
        [193].S.BITS1.27   // 7-DOS-1170-10 FV0
        [193].S.BITS1.28   // 7-DOS-1170-10 FATO
        [193].S.BITS1.30   // 7-DOS-1170-10 Falla Partida
        [193].S.BITS2.27   // 7-DOS-1170-10 Cmd. Marcha
        [193].S.BITS2.20   // 7-DOS-1170-10 Reset Falla
        [193].S.BITS2.23   // 7-DOS-1170-10 Test
        [193].S.BITS2.30   // 7-DOS-1170-10 OUT MARCHA
        [194].S.BITS1.8   // 7-DOS-1170-11 LL
        [194].S.BITS1.9   // 7-DOS-1170-11 LM
        [194].S.BITS1.10   // 7-DOS-1170-11 LH
        [195].S.BITS1.0   // 7-DOS-1170-11 Enable
        [195].S.BITS1.1   // 7-DOS-1170-11 Falla Resumen
        [195].S.BITS1.2   // 7-DOS-1170-11 Conf. Marcha
        [195].S.BITS1.4   // 7-DOS-1170-11 Cmd. Automatico
        [195].S.BITS1.26   // 7-DOS-1170-11 FLL
        [195].S.BITS1.27   // 7-DOS-1170-11 FV0
        [195].S.BITS1.28   // 7-DOS-1170-11 FATO
        [195].S.BITS1.30   // 7-DOS-1170-11 Falla Partida
        [195].S.BITS2.27   // 7-DOS-1170-11 Cmd. Marcha
        [195].S.BITS2.20   // 7-DOS-1170-11 Reset Falla
        [195].S.BITS2.23   // 7-DOS-1170-11 Test
        [195].S.BITS2.30   // 7-DOS-1170-11 OUT MARCHA
        [197].S.BITS1.0   // 7-DOS-1170-12 Enable
        [197].S.BITS1.1   // 7-DOS-1170-12 Falla Resumen
        [197].S.BITS1.2   // 7-DOS-1170-12 Conf. Marcha
        [197].S.BITS1.4   // 7-DOS-1170-12 Cmd. Automatico
        [197].S.BITS1.26   // 7-DOS-1170-12 FLL
        [197].S.BITS1.27   // 7-DOS-1170-12 FV0
        [197].S.BITS1.28   // 7-DOS-1170-12 FATO
        [197].S.BITS1.30   // 7-DOS-1170-12 Falla Partida
        [197].S.BITS2.27   // 7-DOS-1170-12 Cmd. Marcha
        [197].S.BITS2.20   // 7-DOS-1170-12 Reset Falla
        [197].S.BITS2.23   // 7-DOS-1170-12 Test
        [197].S.BITS2.30   // 7-DOS-1170-12 OUT MARCHA
        [201].S.BITS1.0   // 7-DOS-1170a Enable
        [201].S.BITS1.1   // 7-DOS-1170a Falla Resumen
        [201].S.BITS1.2   // 7-DOS-1170a Conf Pos Abrir
        [201].S.BITS1.4   // 7-DOS-1170a Conf Pos Cerrar
        [201].S.BITS1.29   // 7-DOS-1170a Falla Abrir
        [201].S.BITS2.20   // 7-DOS-1170a Reset Falla
        [201].S.BITS2.23   // 7-DOS-1170a Test
        [201].S.BITS2.31   // 7-DOS-1170a OUT OPEN
        [206].S.BITS1.0   // 7-FIL-1173 Enable
        [206].S.BITS1.1   // 7-FIL-1173 Falla Resumen
        [206].S.BITS1.2   // 7-FIL-1173 Conf. Marcha
        [206].S.BITS1.4   // 7-FIL-1173 Cmd. Automatico
        [206].S.BITS1.26   // 7-FIL-1173 FLL
        [206].S.BITS1.27   // 7-FIL-1173 FV0
        [206].S.BITS1.28   // 7-FIL-1173 FATO
        [206].S.BITS1.30   // 7-FIL-1173 Falla Partida
        [206].S.BITS2.27   // 7-FIL-1173 Cmd. Marcha
        [206].S.BITS2.20   // 7-FIL-1173 Reset Falla
        [206].S.BITS2.23   // 7-FIL-1173 Test
        [206].S.BITS2.30   // 7-FIL-1173 OUT MARCHA
        [207].S.BITS1.0   // 7-BBA-1174 Enable
        [207].S.BITS1.1   // 7-BBA-1174 Falla Resumen
        [207].S.BITS1.2   // 7-BBA-1174 Conf. Marcha
        [207].S.BITS1.4   // 7-BBA-1174 Cmd. Automatico
        [207].S.BITS1.26   // 7-BBA-1174 FLL
        [207].S.BITS1.27   // 7-BBA-1174 FV0
        [207].S.BITS1.28   // 7-BBA-1174 FATO
        [207].S.BITS1.30   // 7-BBA-1174 Falla Partida
        [207].S.BITS2.27   // 7-BBA-1174 Cmd. Marcha
        [207].S.BITS2.20   // 7-BBA-1174 Reset Falla
        [207].S.BITS2.23   // 7-BBA-1174 Test
        [207].S.BITS2.30   // 7-BBA-1174 OUT MARCHA
        [215].S.BITS1.0   // 7-BBA-1179a Enable
        [215].S.BITS1.1   // 7-BBA-1179a Falla Resumen
        [215].S.BITS1.2   // 7-BBA-1179a Conf. Marcha
        [215].S.BITS1.4   // 7-BBA-1179a Cmd. Automatico
        [215].S.BITS1.26   // 7-BBA-1179a FLL
        [215].S.BITS1.27   // 7-BBA-1179a FV0
        [215].S.BITS1.28   // 7-BBA-1179a FATO
        [215].S.BITS1.30   // 7-BBA-1179a Falla Partida
        [215].S.BITS2.27   // 7-BBA-1179a Cmd. Marcha
        [215].S.BITS2.20   // 7-BBA-1179a Reset Falla
        [215].S.BITS2.23   // 7-BBA-1179a Test
        [215].S.BITS2.30   // 7-BBA-1179a OUT MARCHA
        [216].S.BITS1.0   // 7-VLV-1179a Enable
        [216].S.BITS1.1   // 7-VLV-1179a Falla Resumen
        [216].S.BITS1.2   // 7-VLV-1179a Conf. Marcha
        [216].S.BITS1.4   // 7-VLV-1179a Cmd. Automatico
        [216].S.BITS1.26   // 7-VLV-1179a FLL
        [216].S.BITS1.27   // 7-VLV-1179a FV0
        [216].S.BITS1.28   // 7-VLV-1179a FATO
        [216].S.BITS1.30   // 7-VLV-1179a Falla Partida
        [216].S.BITS2.27   // 7-VLV-1179a Cmd. Marcha
        [216].S.BITS2.20   // 7-VLV-1179a Reset Falla
        [216].S.BITS2.23   // 7-VLV-1179a Test
        [216].S.BITS2.30   // 7-VLV-1179a OUT MARCHA
        [219].S.BITS1.0   // 7-VLV-1179b Enable
        [219].S.BITS1.1   // 7-VLV-1179b Falla Resumen
        [219].S.BITS1.2   // 7-VLV-1179b Conf. Marcha
        [219].S.BITS1.4   // 7-VLV-1179b Cmd. Automatico
        [219].S.BITS1.26   // 7-VLV-1179b FLL
        [219].S.BITS1.27   // 7-VLV-1179b FV0
        [219].S.BITS1.28   // 7-VLV-1179b FATO
        [219].S.BITS1.30   // 7-VLV-1179b Falla Partida
        [219].S.BITS2.27   // 7-VLV-1179b Cmd. Marcha
        [219].S.BITS2.20   // 7-VLV-1179b Reset Falla
        [219].S.BITS2.23   // 7-VLV-1179b Test
        [219].S.BITS2.30   // 7-VLV-1179b OUT MARCHA
        [221].S.BITS1.0   // 7-BBA-1179c Enable
        [221].S.BITS1.1   // 7-BBA-1179c Falla Resumen
        [221].S.BITS1.2   // 7-BBA-1179c Conf. Marcha
        [221].S.BITS1.4   // 7-BBA-1179c Cmd. Automatico
        [221].S.BITS1.26   // 7-BBA-1179c FLL
        [221].S.BITS1.27   // 7-BBA-1179c FV0
        [221].S.BITS1.28   // 7-BBA-1179c FATO
        [221].S.BITS1.30   // 7-BBA-1179c Falla Partida
        [221].S.BITS2.27   // 7-BBA-1179c Cmd. Marcha
        [221].S.BITS2.20   // 7-BBA-1179c Reset Falla
        [221].S.BITS2.23   // 7-BBA-1179c Test
        [221].S.BITS2.30   // 7-BBA-1179c OUT MARCHA
        [222].S.BITS1.0   // 7-VLV-1179c Enable
        [222].S.BITS1.1   // 7-VLV-1179c Falla Resumen
        [222].S.BITS1.2   // 7-VLV-1179c Conf. Marcha
        [222].S.BITS1.4   // 7-VLV-1179c Cmd. Automatico
        [222].S.BITS1.26   // 7-VLV-1179c FLL
        [222].S.BITS1.27   // 7-VLV-1179c FV0
        [222].S.BITS1.28   // 7-VLV-1179c FATO
        [222].S.BITS1.30   // 7-VLV-1179c Falla Partida
        [222].S.BITS2.27   // 7-VLV-1179c Cmd. Marcha
        [222].S.BITS2.20   // 7-VLV-1179c Reset Falla
        [222].S.BITS2.23   // 7-VLV-1179c Test
        [222].S.BITS2.30   // 7-VLV-1179c OUT MARCHA
        [224].S.BITS1.0   // 7-VIB-1180 Enable
        [224].S.BITS1.1   // 7-VIB-1180 Falla Resumen
        [224].S.BITS1.2   // 7-VIB-1180 Conf. Marcha
        [224].S.BITS1.4   // 7-VIB-1180 Cmd. Automatico
        [224].S.BITS1.26   // 7-VIB-1180 FLL
        [224].S.BITS1.27   // 7-VIB-1180 FV0
        [224].S.BITS1.28   // 7-VIB-1180 FATO
        [224].S.BITS1.30   // 7-VIB-1180 Falla Partida
        [224].S.BITS2.27   // 7-VIB-1180 Cmd. Marcha
        [224].S.BITS2.20   // 7-VIB-1180 Reset Falla
        [224].S.BITS2.23   // 7-VIB-1180 Test
        [224].S.BITS2.30   // 7-VIB-1180 OUT MARCHA
        [228].S.BITS1.0   // 7-RED-1182 Enable
        [228].S.BITS1.1   // 7-RED-1182 Falla Resumen
        [228].S.BITS1.2   // 7-RED-1182 Conf. Marcha
        [228].S.BITS1.4   // 7-RED-1182 Cmd. Automatico
        [228].S.BITS1.26   // 7-RED-1182 FLL
        [228].S.BITS1.27   // 7-RED-1182 FV0
        [228].S.BITS1.28   // 7-RED-1182 FATO
        [228].S.BITS1.30   // 7-RED-1182 Falla Partida
        [228].S.BITS2.27   // 7-RED-1182 Cmd. Marcha
        [228].S.BITS2.20   // 7-RED-1182 Reset Falla
        [228].S.BITS2.23   // 7-RED-1182 Test
        [228].S.BITS2.30   // 7-RED-1182 OUT MARCHA
        [230].S.BITS1.0   // 7-RED-1184 Enable
        [230].S.BITS1.1   // 7-RED-1184 Falla Resumen
        [230].S.BITS1.2   // 7-RED-1184 Conf. Marcha
        [230].S.BITS1.4   // 7-RED-1184 Cmd. Automatico
        [230].S.BITS1.26   // 7-RED-1184 FLL
        [230].S.BITS1.27   // 7-RED-1184 FV0
        [230].S.BITS1.28   // 7-RED-1184 FATO
        [230].S.BITS1.30   // 7-RED-1184 Falla Partida
        [230].S.BITS2.27   // 7-RED-1184 Cmd. Marcha
        [230].S.BITS2.20   // 7-RED-1184 Reset Falla
        [230].S.BITS2.23   // 7-RED-1184 Test
        [230].S.BITS2.30   // 7-RED-1184 OUT MARCHA
        [232].S.BITS1.0   // 7-LMG-1186 Enable
        [232].S.BITS1.1   // 7-LMG-1186 Falla Resumen
        [232].S.BITS1.2   // 7-LMG-1186 Conf Pos Abrir
        [232].S.BITS1.4   // 7-LMG-1186 Conf Pos Cerrar
        [232].S.BITS1.29   // 7-LMG-1186 Falla Abrir
        [232].S.BITS1.30   // 7-LMG-1186 Falla Cerrar
        [232].S.BITS2.20   // 7-LMG-1186 Reset Falla
        [232].S.BITS2.23   // 7-LMG-1186 Test
        [232].S.BITS2.27   // 7-LMG-1186 Cmd. Open
        [232].S.BITS2.30   // 7-LMG-1186 OUT CLOSE
        [232].S.BITS2.31   // 7-LMG-1186 OUT OPEN
        [235].S.BITS2.27   // 7-LRT-1189 Cmd. Marcha
        [237].S.BITS1.0   // 7-RED-1191 Enable
        [237].S.BITS1.1   // 7-RED-1191 Falla Resumen
        [237].S.BITS1.2   // 7-RED-1191 Conf. Marcha
        [237].S.BITS1.4   // 7-RED-1191 Cmd. Automatico
        [237].S.BITS1.26   // 7-RED-1191 FLL
        [237].S.BITS1.27   // 7-RED-1191 FV0
        [237].S.BITS1.28   // 7-RED-1191 FATO
        [237].S.BITS1.30   // 7-RED-1191 Falla Partida
        [237].S.BITS2.27   // 7-RED-1191 Cmd. Marcha
        [237].S.BITS2.20   // 7-RED-1191 Reset Falla
        [237].S.BITS2.23   // 7-RED-1191 Test
        [237].S.BITS2.30   // 7-RED-1191 OUT MARCHA
        [239].S.BITS1.2   // 7-CON-1192 Conf Pos Abrir
        [239].S.BITS1.29   // 7-CON-1192 Falla Abrir
        [240].S.BITS1.0   // 7-CON-1193 Enable
        [240].S.BITS1.1   // 7-CON-1193 Falla Resumen
        [240].S.BITS1.2   // 7-CON-1193 Conf Pos Abrir
        [240].S.BITS1.4   // 7-CON-1193 Conf Pos Cerrar
        [240].S.BITS1.29   // 7-CON-1193 Falla Abrir
        [240].S.BITS1.30   // 7-CON-1193 Falla Cerrar
        [240].S.BITS2.20   // 7-CON-1193 Reset Falla
        [240].S.BITS2.23   // 7-CON-1193 Test
        [240].S.BITS2.27   // 7-CON-1193 Cmd. Open
        [240].S.BITS2.30   // 7-CON-1193 OUT CLOSE
        [240].S.BITS2.31   // 7-CON-1193 OUT OPEN
        [241].S.BITS1.0   // 7-CON-1194 Enable
        [241].S.BITS1.1   // 7-CON-1194 Falla Resumen
        [241].S.BITS1.2   // 7-CON-1194 Conf Pos Abrir
        [241].S.BITS1.4   // 7-CON-1194 Conf Pos Cerrar
        [241].S.BITS1.29   // 7-CON-1194 Falla Abrir
        [241].S.BITS1.30   // 7-CON-1194 Falla Cerrar
        [241].S.BITS2.20   // 7-CON-1194 Reset Falla
        [241].S.BITS2.23   // 7-CON-1194 Test
        [241].S.BITS2.27   // 7-CON-1194 Cmd. Open
        [241].S.BITS2.30   // 7-CON-1194 OUT CLOSE
        [241].S.BITS2.31   // 7-CON-1194 OUT OPEN
        [242].S.BITS1.2   // 7-CON-1195 Conf Pos Abrir
        [245].S.BITS1.26   // 7-ROS-1202 FLL
        [245].S.BITS1.27   // 7-ROS-1202 FV0
        [245].S.BITS1.28   // 7-ROS-1202 FATO
        [245].S.BITS1.30   // 7-ROS-1202 Falla Partida
        [245].S.BITS2.27   // 7-ROS-1202 Cmd. Marcha
        [245].S.BITS2.30   // 7-ROS-1202 OUT MARCHA
        [306].S.BITS1.0   // 8-ROS-610 Enable
        [306].S.BITS1.1   // 8-ROS-610 Falla Resumen
        [306].S.BITS1.2   // 8-ROS-610 Conf. Marcha
        [306].S.BITS1.4   // 8-ROS-610 Cmd. Automatico
        [306].S.BITS1.26   // 8-ROS-610 FLL
        [306].S.BITS1.27   // 8-ROS-610 FV0
        [306].S.BITS1.28   // 8-ROS-610 FATO
        [306].S.BITS1.30   // 8-ROS-610 Falla Partida
        [306].S.BITS2.27   // 8-ROS-610 Cmd. Marcha
        [306].S.BITS2.20   // 8-ROS-610 Reset Falla
        [306].S.BITS2.23   // 8-ROS-610 Test
        [306].S.BITS2.30   // 8-ROS-610 OUT MARCHA
        [309].S.BITS1.0   // 8-ACO-616 Enable
        [309].S.BITS1.1   // 8-ACO-616 Falla Resumen
        [309].S.BITS1.2   // 8-ACO-616 Conf. Marcha
        [309].S.BITS1.4   // 8-ACO-616 Cmd. Automatico
        [309].S.BITS1.26   // 8-ACO-616 FLL
        [309].S.BITS1.27   // 8-ACO-616 FV0
        [309].S.BITS1.28   // 8-ACO-616 FATO
        [309].S.BITS1.30   // 8-ACO-616 Falla Partida
        [309].S.BITS2.27   // 8-ACO-616 Cmd. Marcha
        [309].S.BITS2.20   // 8-ACO-616 Reset Falla
        [309].S.BITS2.23   // 8-ACO-616 Test
        [309].S.BITS2.30   // 8-ACO-616 OUT MARCHA
        [310].S.BITS1.0   // 8-FPR-618 Enable
        [310].S.BITS1.1   // 8-FPR-618 Falla Resumen
        [310].S.BITS1.2   // 8-FPR-618 Conf. Marcha
        [310].S.BITS1.4   // 8-FPR-618 Cmd. Automatico
        [310].S.BITS1.26   // 8-FPR-618 FLL
        [310].S.BITS1.27   // 8-FPR-618 FV0
        [310].S.BITS1.28   // 8-FPR-618 FATO
        [310].S.BITS1.30   // 8-FPR-618 Falla Partida
        [310].S.BITS2.27   // 8-FPR-618 Cmd. Marcha
        [310].S.BITS2.20   // 8-FPR-618 Reset Falla
        [310].S.BITS2.23   // 8-FPR-618 Test
        [310].S.BITS2.30   // 8-FPR-618 OUT MARCHA
        [312].S.BITS1.2   // 8-BIF-624 Conf. Pos. Izquierda
        [312].S.BITS1.4   // 8-BIF-624 Conf. Pos. Derecha
        [312].S.BITS1.29   // 8-BIF-624 Falla Pos. Izquierda
        [312].S.BITS1.30   // 8-BIF-624 Falla Pos. Derecha
        [312].S.BITS2.26   // 8-BIF-624 Cmd. Pos . Izquierda
        [312].S.BITS2.27   // 8-BIF-624 Cmd. Pos. Derecha
        [312].S.BITS2.30   // 8-BIF-624 Out Izquierda
        [319].S.BITS1.8   // 8-CIC-634 LL
        [319].S.BITS1.9   // 8-CIC-634 LM
        [319].S.BITS1.10   // 8-CIC-634 LH
        [324].S.BITS1.0   // 8-VRT-639 Enable
        [324].S.BITS1.1   // 8-VRT-639 Falla Resumen
        [324].S.BITS1.4   // 8-VRT-639 Cmd. Automatico
        [324].S.BITS1.26   // 8-VRT-639 FLL
        [324].S.BITS1.27   // 8-VRT-639 FV0
        [324].S.BITS1.28   // 8-VRT-639 FATO
        [324].S.BITS1.30   // 8-VRT-639 Falla Partida
        [324].S.BITS2.27   // 8-VRT-639 Cmd. Marcha
        [324].S.BITS2.20   // 8-VRT-639 Reset Falla
        [324].S.BITS2.23   // 8-VRT-639 Test
        [324].S.BITS2.30   // 8-VRT-639 OUT MARCHA
        [327].S.BITS1.0   // 8-ENF-640-2 Enable
        [327].S.BITS1.1   // 8-ENF-640-2 Falla Resumen
        [327].S.BITS1.2   // 8-ENF-640-2 Conf. Marcha
        [327].S.BITS1.4   // 8-ENF-640-2 Cmd. Automatico
        [327].S.BITS1.30   // 8-ENF-640-2 Falla Partida
        [327].S.BITS2.27   // 8-ENF-640-2 Cmd. Marcha
        [327].S.BITS2.20   // 8-ENF-640-2 Reset Falla
        [327].S.BITS2.23   // 8-ENF-640-2 Test
        [327].S.BITS2.30   // 8-ENF-640-2 OUT MARCHA
        [329].S.BITS1.8   // 8-CIC-644 LL
        [329].S.BITS1.9   // 8-CIC-644 LM
        [329].S.BITS1.10   // 8-CIC-644 LH
        [330].S.BITS1.0   // 8-VRT-648 Enable
        [330].S.BITS1.1   // 8-VRT-648 Falla Resumen
        [330].S.BITS1.2   // 8-VRT-648 Conf. Marcha
        [330].S.BITS1.4   // 8-VRT-648 Cmd. Automatico
        [330].S.BITS1.26   // 8-VRT-648 FLL
        [330].S.BITS1.27   // 8-VRT-648 FV0
        [330].S.BITS1.28   // 8-VRT-648 FATO
        [330].S.BITS1.30   // 8-VRT-648 Falla Partida
        [330].S.BITS2.27   // 8-VRT-648 Cmd. Marcha
        [330].S.BITS2.20   // 8-VRT-648 Reset Falla
        [330].S.BITS2.23   // 8-VRT-648 Test
        [330].S.BITS2.30   // 8-VRT-648 OUT MARCHA
        [339].S.BITS1.30   // 8-ELV-662 Falla Partida
        [339].S.BITS2.27   // 8-ELV-662 Cmd. Marcha
        [339].S.BITS2.30   // 8-ELV-662 OUT MARCHA
        [342].S.BITS1.2   // 8-CON-664b Conf Pos Abrir
        [342].S.BITS1.29   // 8-CON-664b Falla Abrir
        [350].S.BITS1.0   // 8-ROS-714 Enable
        [350].S.BITS1.1   // 8-ROS-714 Falla Resumen
        [350].S.BITS1.2   // 8-ROS-714 Conf. Marcha
        [350].S.BITS1.4   // 8-ROS-714 Cmd. Automatico
        [350].S.BITS1.26   // 8-ROS-714 FLL
        [350].S.BITS1.27   // 8-ROS-714 FV0
        [350].S.BITS1.28   // 8-ROS-714 FATO
        [350].S.BITS1.30   // 8-ROS-714 Falla Partida
        [350].S.BITS2.27   // 8-ROS-714 Cmd. Marcha
        [350].S.BITS2.20   // 8-ROS-714 Reset Falla
        [350].S.BITS2.23   // 8-ROS-714 Test
        [350].S.BITS2.30   // 8-ROS-714 OUT MARCHA
        [354].S.BITS1.2   // 8-BIF-724 Conf. Pos. Izquierda
        [354].S.BITS1.4   // 8-BIF-724 Conf. Pos. Derecha
        [354].S.BITS1.29   // 8-BIF-724 Falla Pos. Izquierda
        [354].S.BITS1.30   // 8-BIF-724 Falla Pos. Derecha
        [354].S.BITS2.26   // 8-BIF-724 Cmd. Pos . Izquierda
        [354].S.BITS2.27   // 8-BIF-724 Cmd. Pos. Derecha
        [354].S.BITS2.30   // 8-BIF-724 Out Izquierda
        [354].S.BITS2.31   // 8-BIF-724 Out Derecha
        [357].S.BITS1.30   // 8-ENF-730-1 Falla Partida
        [357].S.BITS2.27   // 8-ENF-730-1 Cmd. Marcha
        [357].S.BITS2.30   // 8-ENF-730-1 OUT MARCHA
        [358].S.BITS1.8   // 8-ENF-730 LL
        [361].S.BITS1.8   // 8-CIC-734 LL
        [361].S.BITS1.9   // 8-CIC-734 LM
        [361].S.BITS1.10   // 8-CIC-734 LH
        [364].S.BITS1.26   // 8-VEN-737 FLL
        [364].S.BITS1.27   // 8-VEN-737 FV0
        [364].S.BITS1.28   // 8-VEN-737 FATO
        [368].S.BITS1.8   // 8-ENF-740 LL
        [368].S.BITS1.9   // 8-ENF-740 LM
        [368].S.BITS1.10   // 8-ENF-740 LH
        [369].S.BITS1.0   // 8-ENF-740-2 Enable
        [369].S.BITS1.1   // 8-ENF-740-2 Falla Resumen
        [369].S.BITS1.4   // 8-ENF-740-2 Cmd. Automatico
        [369].S.BITS1.26   // 8-ENF-740-2 FLL
        [369].S.BITS1.27   // 8-ENF-740-2 FV0
        [369].S.BITS1.28   // 8-ENF-740-2 FATO
        [369].S.BITS1.30   // 8-ENF-740-2 Falla Partida
        [369].S.BITS2.27   // 8-ENF-740-2 Cmd. Marcha
        [369].S.BITS2.20   // 8-ENF-740-2 Reset Falla
        [369].S.BITS2.23   // 8-ENF-740-2 Test
        [369].S.BITS2.30   // 8-ENF-740-2 OUT MARCHA
        [371].S.BITS1.8   // 8-CIC-744 LL
        [371].S.BITS1.9   // 8-CIC-744 LM
        [371].S.BITS1.10   // 8-CIC-744 LH
        [379].S.BITS1.26   // 8-RED-758 FLL
        [379].S.BITS1.27   // 8-RED-758 FV0
        [379].S.BITS1.28   // 8-RED-758 FATO
        [379].S.BITS2.27   // 8-RED-758 Cmd. Marcha
        [383].S.BITS1.0   // 8-RED-766 Enable
        [383].S.BITS1.1   // 8-RED-766 Falla Resumen
        [383].S.BITS1.2   // 8-RED-766 Conf. Marcha
        [383].S.BITS1.4   // 8-RED-766 Cmd. Automatico
        [383].S.BITS1.26   // 8-RED-766 FLL
        [383].S.BITS1.27   // 8-RED-766 FV0
        [383].S.BITS1.28   // 8-RED-766 FATO
        [383].S.BITS1.30   // 8-RED-766 Falla Partida
        [383].S.BITS2.27   // 8-RED-766 Cmd. Marcha
        [383].S.BITS2.20   // 8-RED-766 Reset Falla
        [383].S.BITS2.23   // 8-RED-766 Test
        [383].S.BITS2.30   // 8-RED-766 OUT MARCHA
        [385].S.BITS1.8   // 8-TOL-800 LL
        [385].S.BITS1.9   // 8-TOL-800 LM
        [385].S.BITS1.10   // 8-TOL-800 LH
        [386].S.BITS2.27   // 9-RED-650 Cmd. Marcha
        [388].S.BITS1.2   // 9-CON-652 Conf Pos Abrir
        [388].S.BITS1.29   // 9-CON-652 Falla Abrir
        [388].S.BITS2.31   // 9-CON-652 OUT OPEN
        [392].S.BITS1.26   // 9-RED-655 FLL
        [392].S.BITS1.27   // 9-RED-655 FV0
        [392].S.BITS1.28   // 9-RED-655 FATO
        [392].S.BITS2.27   // 9-RED-655 Cmd. Marcha
        [393].S.BITS1.0   // 9-CON-656 Enable
        [393].S.BITS1.1   // 9-CON-656 Falla Resumen
        [393].S.BITS1.2   // 9-CON-656 Conf Pos Abrir
        [393].S.BITS1.4   // 9-CON-656 Conf Pos Cerrar
        [393].S.BITS1.29   // 9-CON-656 Falla Abrir
        [393].S.BITS1.30   // 9-CON-656 Falla Cerrar
        [393].S.BITS2.20   // 9-CON-656 Reset Falla
        [393].S.BITS2.23   // 9-CON-656 Test
        [393].S.BITS2.27   // 9-CON-656 Cmd. Open
        [393].S.BITS2.30   // 9-CON-656 OUT CLOSE
        [393].S.BITS2.31   // 9-CON-656 OUT OPEN
        [394].S.BITS1.2   // 9-CON-657 Conf Pos Abrir
        [394].S.BITS1.29   // 9-CON-657 Falla Abrir
        [394].S.BITS2.31   // 9-CON-657 OUT OPEN
        [396].S.BITS1.0   // 9-CON-659 Enable
        [396].S.BITS1.1   // 9-CON-659 Falla Resumen
        [396].S.BITS1.2   // 9-CON-659 Conf Pos Abrir
        [396].S.BITS1.4   // 9-CON-659 Conf Pos Cerrar
        [396].S.BITS1.29   // 9-CON-659 Falla Abrir
        [396].S.BITS1.30   // 9-CON-659 Falla Cerrar
        [396].S.BITS2.20   // 9-CON-659 Reset Falla
        [396].S.BITS2.23   // 9-CON-659 Test
        [396].S.BITS2.27   // 9-CON-659 Cmd. Open
        [396].S.BITS2.30   // 9-CON-659 OUT CLOSE
        [396].S.BITS2.31   // 9-CON-659 OUT OPEN
        [398].S.BITS1.26   // 9-RED-660 FLL
        [398].S.BITS1.27   // 9-RED-660 FV0
        [398].S.BITS1.28   // 9-RED-660 FATO
        [398].S.BITS2.27   // 9-RED-660 Cmd. Marcha
        [400].S.BITS1.2   // 9-CON-662 Conf Pos Abrir
        [400].S.BITS1.29   // 9-CON-662 Falla Abrir
        [400].S.BITS2.31   // 9-CON-662 OUT OPEN
        [406].S.BITS1.2   // 9-CON-668 Conf Pos Abrir
        [406].S.BITS1.29   // 9-CON-668 Falla Abrir
        [406].S.BITS2.31   // 9-CON-668 OUT OPEN
        [408].S.BITS1.26   // 9-RED-670 FLL
        [408].S.BITS1.27   // 9-RED-670 FV0
        [408].S.BITS1.28   // 9-RED-670 FATO
        [408].S.BITS2.27   // 9-RED-670 Cmd. Marcha
        [414].S.BITS1.29   // 9-CON-676 Falla Abrir
        [421].S.BITS1.2   // 9-CON-683 Conf Pos Abrir
        [433].S.BITS1.29   // 9-CON-695 Falla Abrir
        [443].S.BITS1.2   // 9-CON-705 Conf Pos Abrir
        [448].S.BITS1.8   // 9-BIN-710 LL
        [448].S.BITS1.9   // 9-BIN-710 LM
        [448].S.BITS1.10   // 9-BIN-710 LH
        [451].S.BITS1.29   // 9-CON-713 Falla Abrir
        [452].S.BITS1.8   // 9-BIN-714 LL
        [452].S.BITS1.9   // 9-BIN-714 LM
        [452].S.BITS1.10   // 9-BIN-714 LH
        [454].S.BITS1.8   // 9-BIN-716 LL
        [454].S.BITS1.9   // 9-BIN-716 LM
        [454].S.BITS1.10   // 9-BIN-716 LH
        [456].S.BITS1.8   // 9-BIN-718 LL
        [456].S.BITS1.9   // 9-BIN-718 LM
        [456].S.BITS1.10   // 9-BIN-718 LH
        [458].S.BITS1.8   // 9-BIN-720 LL
        [458].S.BITS1.9   // 9-BIN-720 LM
        [458].S.BITS1.10   // 9-BIN-720 LH
        [460].S.BITS1.8   // 9-BIN-722 LL
        [460].S.BITS1.9   // 9-BIN-722 LM
        [460].S.BITS1.10   // 9-BIN-722 LH
        [468].S.BITS1.8   // 9-BIN-730 LL
        [468].S.BITS1.9   // 9-BIN-730 LM
        [468].S.BITS1.10   // 9-BIN-730 LH
   _Eqp_Cfg : Eqp_Cfg[800] := ([1].Type := 2, [2].Type := 256, [3].Type := 2, [3].Setup := 98, [4].Type := 2, [4].Setup := 66, [5].Type := 2, [6].Type := 8, [7].Type := 128, [7].Setup := 16400, [8].Type := 128, [8].Setup := 16400, [10].Type := 64, [10].Setup := 80, [11].Type := 64, [11].Setup := 80, [12].Type := 64, [12].Setup := 80, [13].Type := 64, [13].Setup := 80, [14].Type := 64, [14].Setup := 80, [15].Type := 64, [15].Setup := 80, [20].Type := 256, [21].Type := 256, [22].Type := 256, [23].Type := 256, [24].Type := 256, [25].Type := 256, [26].Type := 256, [27].Type := 256, [28].Type := 256, [29].Type := 256, [30].Type := 256, [31].Type := 256, [32].Type := 256, [33].Type := 256, [34].Type := 256, [35].Type := 256, [40].Type := 2, [40].Setup := 114, [41].Type := 2, [41].Setup := 114, [42].Type := 2, [42].Setup := 114, [43].Type := 2, [43].Setup := 114, [44].Type := 2, [44].Setup := 114, [45].Type := 2, [45].Setup := 114, [46].Type := 2, [46].Setup := 114, [47].Type := 2, [47].Setup := 114, [48].Type := 2, [48].Setup := 114, [49].Type := 2, [49].Setup := 114,
        [50].Type := 2, [50].Setup := 114, [51].Type := 2, [51].Setup := 114, [52].Type := 2, [52].Setup := 114, [53].Type := 2, [53].Setup := 114, [54].Type := 2, [54].Setup := 114, [55].Type := 2, [55].Setup := 114, [60].Type := 256, [61].Type := 256, [62].Type := 256, [63].Type := 256, [64].Type := 256, [65].Type := 256, [66].Type := 256, [67].Type := 256, [68].Type := 256, [69].Type := 256, [70].Type := 256, [71].Type := 256, [72].Type := 256, [73].Type := 256, [74].Type := 256, [74].Setup := 96, [80].Type := 2, [80].Setup := 114, [81].Type := 2, [81].Setup := 114, [82].Type := 2, [82].Setup := 114, [83].Type := 2, [83].Setup := 114, [84].Type := 2, [84].Setup := 114, [85].Type := 2, [85].Setup := 114, [86].Type := 2, [86].Setup := 114, [87].Type := 2, [87].Setup := 114, [88].Type := 2, [88].Setup := 114, [89].Type := 2, [89].Setup := 114, [90].Type := 2, [90].Setup := 114, [91].Type := 2, [91].Setup := 114, [92].Type := 2, [92].Setup := 114, [93].Type := 2, [93].Setup := 114, [94].Type := 64, [94].Setup := 114, [100].Type := 64, [100].Setup := 80,
        [101].Type := 64, [101].Setup := 80, [102].Type := 64, [102].Setup := 80, [103].Type := 64, [103].Setup := 80, [104].Type := 64, [104].Setup := 80, [105].Type := 64, [105].Setup := 80, [110].Type := 256, [111].Type := 64, [111].Setup := 114, [112].Type := 256, [113].Type := 64, [113].Setup := 114, [114].Type := 256, [115].Type := 64, [115].Setup := 114, [116].Type := 256, [117].Type := 64, [117].Setup := 114, [118].Type := 64, [118].Setup := 82, [119].Type := 64, [119].Setup := 82, [120].Type := 256, [121].Type := 64, [121].Setup := 80, [123].Type := 2, [123].Setup := 114, [129].Type := 256, [130].Type := 2, [130].Setup := 64, [131].Type := 64, [131].Setup := 98, [132].Type := 256, [133].Type := 2, [133].Setup := 96, [134].Type := 2, [134].Setup := 64, [135].Type := 2, [136].Type := 2, [137].Type := 2, [137].Setup := 64, [138].Type := 8, [140].Type := 256, [141].Type := 64, [141].Setup := 96, [150].Type := 256, [151].Type := 64, [151].Setup := 96, [152].Type := 256, [153].Type := 64, [153].Setup := 608, [154].Type := 64, [154].Setup := 608, [155].Type := 64, [155].Setup := 608, [156].Type := 64,
        [156].Setup := 608, [157].Type := 64, [157].Setup := 608, [158].Type := 64, [158].Setup := 608, [159].Type := 64, [159].Setup := 608, [160].Type := 64, [160].Setup := 608, [161].Type := 64, [161].Setup := 608, [162].Type := 64, [162].Setup := 608, [163].Type := 64, [163].Setup := 608, [164].Type := 64, [164].Setup := 608, [165].Type := 64, [165].Setup := 608, [166].Type := 64, [166].Setup := 608, [167].Type := 64, [167].Setup := 608, [168].Type := 64, [168].Setup := 608, [170].Type := 1073741824, [170].Setup := 64, [171].Type := 1073741824, [171].Setup := 64);
   _Origen : Origen[40] := ([1]._1eqp := 3, [1].Color := 3, [1].DestReal := 26, [1].DestOld := 26, [1].DestNew := 7, [1].Prod1eqpInd := 51, [1].ProdFinInd := 51, [1].Tespera.PRE := 120000, [2]._1eqp := 133, [2].Bits := 1, [2].Color := 6, [2].DestReal := 150, [2].DestOld := 150, [2].DestNew := 2, [2].Tespera.PRE := 120000, [3]._1eqp := 29, [3].Color := 5, [3].DestReal := 119, [3].DestOld := 119, [3].DestNew := 3, [3].Prod1eqpInd := 428, [3].ProdFinInd := 428, [3].Tespera.PRE := 120000, [4]._1eqp := 141, [4].Color := 5, [4].DestReal := 158, [4].DestOld := 158, [4].DestNew := 2, [4].Prod1eqpInd := 49, [4].ProdFinInd := 49, [4].Tespera.PRE := 120000, [5]._1eqp := 45, [5].Color := 3, [5].DestReal := 44, [5].DestOld := 44, [5].DestNew := 1, [5].Prod1eqpInd := 7, [5].ProdFinInd := 7, [5].Tespera.PRE := 120000, [6]._1eqp := 58, [6].Color := 4, [6].DestReal := 107, [6].DestOld := 107, [6].DestNew := 1, [6].Prod1eqpInd := 2081, [6].ProdFinInd := 2081, [6].Tespera.PRE := 120000, [7]._1eqp := 77, [7].Color := 4, [7].DestReal := 107, [7].DestOld := 107, [7].DestNew := 1, [7].Prod1eqpInd := 2081, [7].ProdFinInd := 2081, [7].Tespera.PRE := 120000, [8]._1eqp := 227, [8].Color := 5, [8].DestReal := 301, [8].DestOld := 301, [8].DestNew := 1,
        [8].Tespera.PRE := 120000, [9]._1eqp := 306, [9].Color := 3, [9].Tespera.PRE := 120000, [10]._1eqp := 348, [10].Color := 5, [10].Tespera.PRE := 120000, [11]._1eqp := 337, [11].Color := 5, [11].DestReal := 446, [11].DestOld := 446, [11].DestNew := 5, [11].Prod1eqpInd := 6704, [11].ProdFinInd := 6704, [11].Tespera.PRE := 120000, [12]._1eqp := 379, [12].Color := 4, [12].DestReal := 442, [12].DestOld := 442, [12].DestNew := 3, [12].Prod1eqpInd := 6706, [12].ProdFinInd := 6706, [12].Tespera.PRE := 120000, [13]._1eqp := 262, [13].Color := 3, [13].DestReal := 44, [13].DestOld := 44, [13].DestNew := 1, [13].Prod1eqpInd := 7, [13].ProdFinInd := 7, [13].Tespera.PRE := 120000, [14]._1eqp := 48, [14].Color := 3, [14].DestReal := 115, [14].DestOld := 115, [14].DestNew := 6, [14].Prod1eqpInd := 7, [14].ProdFinInd := 7, [14].Tespera.PRE := 120000, [15]._1eqp := 250, [15].Bits := 16, [15].DestNew := 2, [15].Tespera.PRE := 120000, [16]._1eqp := 379, [16].Color := 4, [16].Tespera.PRE := 120000, [17]._1eqp := 29, [17].Bits := 16, [17].DestReal := 123, [17].DestOld := 123, [17].DestNew := 7, [17].Tespera.PRE := 120000, [18]._1eqp := 250, [18].DestReal := 123, [18].DestOld := 123, [18].DestNew := 5, [18].Tespera.PRE := 120000);
        [1].BITS.0   // Start Ruta 1
        [1].BITS.2   // Cambio Ruta 1
        [2].BITS.0   // Start Ruta 2
        [2].BITS.2   // Cambio Ruta 2
        [3].BITS.0   // Origen RED-046-00
        [3].BITS.2   // Origen RED-046-00
        [1].BITS.7   // Deshabilitar Cambio de Ruta con carga
   _Parametros_D : DINT[30] := ([0] := 60, [1] := 30, [2] := 40);
        [0]   // Tiempo de Mezcla [s]
        [1]   // Tiempo de Mezcla (Ingr.) [s]
        [2]   // Tiempo Arriba Transporte [s]
   _Parametros_F : REAL[30] := ([0] := 5.0, [1] := 1.0, [2] := 0.05, [3] := 0.05, [4] := 15.0, [5] := 9.0, [6] := 17.0, [7] := 7.0, [8] := 16.0);
        [0]   // Peso Vacío Macros
        [1]   // Peso Vacío Midis
        [2]   // Peso Vacío Micros 1
        [3]   // Peso Vacío Micros 2
        [4]   // Corriente de Vacío Mezcladora
        [5]   // Corriente de Vacío Elevador a Despacho
        [6]   // Corriente de Carga Elevador a Despacho
        [7]   // Corriente Vacío Elevador Abastecimiento
        [8]   // Corriente Carga Elevador Abastecimiento
   _reset_locales : DINT;
        .0   // Reset local DB
        .1   // Reset local Gestion Dosificación
   _SS : Soft_Starter[20] := ([1].Idx_Equipo[0] := 106, [1].Idx_Equipo[1] := 107, [1].Idx_Equipo[2] := 108, [1].Idx_Equipo[3] := 109, [1].Partiendo := 1, [1].Flags := 1, [1].Tpo_Espera.PRE := 15000, [1].Tpos_Grl[0].PRE := 3000, [2].Idx_Equipo[0] := 63, [2].Idx_Equipo[1] := 64, [2].Idx_Equipo[2] := 65, [2].Partiendo := 1, [2].Flags := 1, [2].Tpo_Espera.PRE := 15000, [2].Tpos_Grl[0].PRE := 3000, [3].Idx_Equipo[0] := 73, [3].Idx_Equipo[1] := 74, [3].Idx_Equipo[2] := 75, [3].Partiendo := 1, [3].Flags := 1, [3].Tpo_Espera.PRE := 15000, [3].Tpos_Grl[0].PRE := 3000, [4].Idx_Equipo[0] := 83, [4].Idx_Equipo[1] := 84, [4].Idx_Equipo[2] := 85, [4].Partiendo := 1, [4].Flags := 1, [4].Tpo_Espera.PRE := 15000, [4].Tpos_Grl[0].PRE := 3000, [5].Idx_Equipo[0] := 45, [5].Idx_Equipo[1] := 92, [5].Idx_Equipo[2] := 103, [5].Idx_Equipo[3] := 26, [5].Idx_Equipo[4] := 28, [5].Partiendo := 1, [5].Flags := 1, [5].Tpo_Espera.PRE := 15000, [5].Tpos_Grl[0].PRE := 3000, [6].Idx_Equipo[0] := 326, [6].Idx_Equipo[1] := 325, [6].Partiendo := 1, [6].Flags := 1, [6].Tpo_Espera.PRE := 15000, [6].Tpos_Grl[0].PRE := 3000, [7].Idx_Equipo[0] := 554, [7].Idx_Equipo[1] := 574, [7].Idx_Equipo[2] := 524, [7].Idx_Equipo[3] := 372, [7].Idx_Equipo[4] := 502, [7].Eqp_Actual := 564, [7].Partiendo := 1, [7].Flags := 2, [7].Tpo_Espera.PRE := 15000, [7].Tpos_Grl[0].PRE := 3000, [8].Idx_Equipo[0] := 283, [8].Eqp_Actual := 554, [8].Disponible := 1, [8].Tpo_Espera.PRE := 15000, [8].Tpos_Grl[0].PRE := 3000, [9].Idx_Equipo[0] := 46,
        [9].Partiendo := 1, [9].Flags := 1, [9].Tpo_Espera.PRE := 15000, [9].Tpos_Grl[0].PRE := 3000, [10].Idx_Equipo[0] := 57, [10].Partiendo := 1, [10].Flags := 1, [10].Tpo_Espera.PRE := 15000, [10].Tpos_Grl[0].PRE := 3000, [11].Idx_Equipo[0] := 322, [11].Partiendo := 1, [11].Flags := 1, [11].Tpo_Espera.PRE := 15000, [11].Tpos_Grl[0].PRE := 3000, [12].Partiendo := 1, [12].Tpo_Espera.PRE := 15000, [12].Tpos_Grl[0].PRE := 3000, [13].Disponible := 1, [13].Tpo_Espera.PRE := 15000, [13].Tpos_Grl[0].PRE := 3000);
   _Typlgie : Eqp_Typologie[800] := ([1].Type := 1, [1].Syst := 1, [1].Area := 1, [2].Type := 8, [2].Syst := 1, [2].Area := 1, [3].Next := 4, [3].Type := 1, [3].Setup := 98, [3].Syst := 1, [3].Area := 1, [3].Indx[3] := 1, [4].Next := 170, [4].Type := 1, [4].Setup := 66, [4].Syst := 1, [4].Area := 1, [5].Type := 1, [5].Syst := 1, [5].Area := 1, [6].Type := 3, [6].Syst := 1, [6].Area := 1, [7].Type := 7, [7].Setup := 16400, [7].Syst := 2, [7].Area := 1, [7].Indx[5] := 8, [7].Indx[6] := 1, [8].Type := 7, [8].Setup := 16400, [8].Syst := 3, [8].Area := 1, [8].Indx[5] := 8, [8].Indx[6] := 2, [10].Next := 110, [10].Type := 6, [10].Setup := 80, [10].Syst := 3, [10].Area := 1, [11].Next := 112, [11].Type := 6, [11].Setup := 80, [11].Syst := 3, [11].Area := 1, [12].Next := 112, [12].Type := 6, [12].Setup := 80, [12].Syst := 3, [12].Area := 1, [13].Next := 110, [13].Type := 6, [13].Setup := 80, [13].Syst := 3, [13].Area := 1, [14].Next := 110, [14].Type := 6, [14].Setup := 80, [14].Syst := 3, [14].Area := 1,
        [15].Next := 112, [15].Type := 6, [15].Setup := 80, [15].Syst := 3, [15].Area := 1, [20].Type := 8, [20].Syst := 2, [20].Area := 1, [20].Indx[3] := 2, [21].Type := 8, [21].Syst := 2, [21].Area := 1, [21].Indx[3] := 3, [22].Type := 8, [22].Syst := 2, [22].Area := 1, [22].Indx[3] := 4, [23].Type := 8, [23].Syst := 2, [23].Area := 1, [23].Indx[3] := 5, [24].Type := 8, [24].Syst := 2, [24].Area := 1, [24].Indx[3] := 6, [25].Type := 8, [25].Syst := 2, [25].Area := 1, [25].Indx[3] := 7, [26].Type := 8, [26].Syst := 2, [26].Area := 1, [26].Indx[3] := 8, [27].Type := 8, [27].Syst := 2, [27].Area := 1, [27].Indx[3] := 9, [28].Type := 8, [28].Syst := 3, [28].Area := 1, [28].Indx[3] := 10, [29].Type := 8, [29].Syst := 3, [29].Area := 1, [29].Indx[3] := 11, [30].Type := 8, [30].Syst := 3, [30].Area := 1, [30].Indx[3] := 12, [31].Type := 8, [31].Syst := 3, [31].Area := 1, [31].Indx[3] := 13, [32].Type := 8, [32].Syst := 3, [32].Area := 1, [32].Indx[3] := 14, [33].Type := 8, [33].Syst := 3, [33].Area := 1,
        [33].Indx[3] := 15, [34].Type := 8, [34].Syst := 3, [34].Area := 1, [34].Indx[3] := 16, [35].Type := 8, [35].Syst := 3, [35].Area := 1, [35].Indx[3] := 17, [40].Next := 110, [40].Type := 1, [40].Setup := 114, [40].Syst := 2, [40].Area := 1, [40].Indx[0] := 1, [40].Indx[1] := 1, [40].Indx[2] := 1, [41].Next := 110, [41].Type := 1, [41].Setup := 114, [41].Syst := 2, [41].Area := 1, [41].Indx[0] := 2, [41].Indx[1] := 1, [41].Indx[2] := 2, [42].Next := 110, [42].Type := 1, [42].Setup := 114, [42].Syst := 2, [42].Area := 1, [42].Indx[0] := 3, [42].Indx[1] := 1, [42].Indx[2] := 3, [43].Next := 10, [43].Type := 1, [43].Setup := 114, [43].Syst := 2, [43].Area := 1, [43].Indx[0] := 4, [43].Indx[1] := 1, [43].Indx[2] := 4, [44].Next := 11, [44].Type := 1, [44].Setup := 114, [44].Syst := 2, [44].Area := 1, [44].Indx[0] := 5, [44].Indx[1] := 2, [44].Indx[2] := 5, [45].Next := 112, [45].Type := 1, [45].Setup := 114, [45].Syst := 2, [45].Area := 1, [45].Indx[0] := 6, [45].Indx[1] := 2, [45].Indx[2] := 6, [46].Next := 12, [46].Type := 1, [46].Setup := 114,
        [46].Syst := 2, [46].Area := 1, [46].Indx[0] := 7, [46].Indx[1] := 2, [46].Indx[2] := 7, [47].Next := 112, [47].Type := 1, [47].Setup := 114, [47].Syst := 2, [47].Area := 1, [47].Indx[0] := 8, [47].Indx[1] := 2, [47].Indx[2] := 8, [48].Next := 110, [48].Type := 1, [48].Setup := 114, [48].Syst := 3, [48].Area := 1, [48].Indx[0] := 9, [48].Indx[1] := 1, [48].Indx[2] := 9, [49].Next := 13, [49].Type := 1, [49].Setup := 114, [49].Syst := 3, [49].Area := 1, [49].Indx[0] := 10, [49].Indx[1] := 1, [49].Indx[2] := 10, [50].Next := 110, [50].Type := 1, [50].Setup := 114, [50].Syst := 3, [50].Area := 1, [50].Indx[0] := 11, [50].Indx[1] := 1, [50].Indx[2] := 11, [51].Next := 14, [51].Type := 1, [51].Setup := 114, [51].Syst := 3, [51].Area := 1, [51].Indx[0] := 12, [51].Indx[1] := 1, [51].Indx[2] := 12, [52].Next := 112, [52].Type := 1, [52].Setup := 114, [52].Syst := 3, [52].Area := 1, [52].Indx[0] := 13, [52].Indx[1] := 2, [52].Indx[2] := 13, [53].Next := 112, [53].Type := 1, [53].Setup := 114, [53].Syst := 3, [53].Area := 1, [53].Indx[0] := 14, [53].Indx[1] := 2,
        [53].Indx[2] := 14, [54].Next := 112, [54].Type := 1, [54].Setup := 114, [54].Syst := 3, [54].Area := 1, [54].Indx[0] := 15, [54].Indx[1] := 2, [54].Indx[2] := 15, [55].Next := 15, [55].Type := 1, [55].Setup := 114, [55].Syst := 3, [55].Area := 1, [55].Indx[0] := 16, [55].Indx[1] := 2, [55].Indx[2] := 16, [60].Type := 8, [60].Syst := 4, [60].Area := 1, [61].Type := 8, [61].Syst := 4, [61].Area := 1, [62].Type := 8, [62].Syst := 4, [62].Area := 1, [63].Type := 8, [63].Syst := 4, [63].Area := 1, [64].Type := 8, [64].Syst := 4, [64].Area := 1, [65].Type := 8, [65].Syst := 4, [65].Area := 1, [66].Type := 8, [66].Syst := 4, [66].Area := 1, [67].Type := 8, [67].Syst := 5, [67].Area := 1, [68].Type := 8, [68].Syst := 5, [68].Area := 1, [69].Type := 8, [69].Syst := 5, [69].Area := 1, [70].Type := 8, [70].Syst := 5, [70].Area := 1, [71].Type := 8, [71].Syst := 5, [71].Area := 1, [72].Type := 8, [72].Syst := 5, [72].Area := 1, [73].Type := 8, [73].Syst := 5, [73].Area := 1, [74].Next := 94,
        [74].Type := 8, [74].Setup := 96, [74].Syst := 5, [74].Area := 1, [80].Next := 114, [80].Type := 1, [80].Setup := 114, [80].Syst := 4, [80].Area := 1, [80].Indx[0] := 17, [80].Indx[1] := 3, [80].Indx[2] := 17, [81].Next := 100, [81].Type := 1, [81].Setup := 114, [81].Syst := 4, [81].Area := 1, [81].Indx[0] := 18, [81].Indx[1] := 3, [81].Indx[2] := 18, [82].Next := 114, [82].Type := 1, [82].Setup := 114, [82].Syst := 4, [82].Area := 1, [82].Indx[0] := 19, [82].Indx[1] := 3, [82].Indx[2] := 19, [83].Next := 101, [83].Type := 1, [83].Setup := 114, [83].Syst := 4, [83].Area := 1, [83].Indx[0] := 20, [83].Indx[1] := 3, [83].Indx[2] := 20, [84].Next := 114, [84].Type := 1, [84].Setup := 114, [84].Syst := 4, [84].Area := 1, [84].Indx[0] := 21, [84].Indx[1] := 3, [84].Indx[2] := 21, [85].Next := 102, [85].Type := 1, [85].Setup := 114, [85].Syst := 4, [85].Area := 1, [85].Indx[0] := 22, [85].Indx[1] := 3, [85].Indx[2] := 22, [86].Next := 114, [86].Type := 1, [86].Setup := 114, [86].Syst := 4, [86].Area := 1, [86].Indx[0] := 23, [86].Indx[1] := 3, [86].Indx[2] := 23,
        [87].Next := 116, [87].Type := 1, [87].Setup := 114, [87].Syst := 5, [87].Area := 1, [87].Indx[0] := 24, [87].Indx[1] := 4, [87].Indx[2] := 24, [88].Next := 103, [88].Type := 1, [88].Setup := 114, [88].Syst := 5, [88].Area := 1, [88].Indx[0] := 25, [88].Indx[1] := 4, [88].Indx[2] := 25, [89].Next := 116, [89].Type := 1, [89].Setup := 114, [89].Syst := 5, [89].Area := 1, [89].Indx[0] := 26, [89].Indx[1] := 4, [89].Indx[2] := 26, [90].Next := 104, [90].Type := 1, [90].Setup := 114, [90].Syst := 5, [90].Area := 1, [90].Indx[0] := 27, [90].Indx[1] := 4, [90].Indx[2] := 27, [91].Next := 116, [91].Type := 1, [91].Setup := 114, [91].Syst := 5, [91].Area := 1, [91].Indx[0] := 28, [91].Indx[1] := 4, [91].Indx[2] := 28, [92].Next := 105, [92].Type := 1, [92].Setup := 114, [92].Syst := 5, [92].Area := 1, [92].Indx[0] := 29, [92].Indx[1] := 4, [92].Indx[2] := 29, [93].Next := 116, [93].Type := 1, [93].Setup := 114, [93].Syst := 5, [93].Area := 1, [93].Indx[0] := 30, [93].Indx[1] := 4, [93].Indx[2] := 30, [94].Next := 119, [94].Type := 6, [94].Setup := 114, [94].Syst := 5,
        [94].Area := 1, [94].Indx[0] := 31, [94].Indx[1] := 5, [94].Indx[2] := 31, [100].Next := 114, [100].Type := 6, [100].Setup := 80, [100].Syst := 4, [100].Area := 1, [101].Next := 114, [101].Type := 6, [101].Setup := 80, [101].Syst := 4, [101].Area := 1, [102].Next := 114, [102].Type := 6, [102].Setup := 80, [102].Syst := 4, [102].Area := 1, [103].Next := 116, [103].Type := 6, [103].Setup := 80, [103].Syst := 5, [103].Area := 1, [104].Next := 116, [104].Type := 6, [104].Setup := 80, [104].Syst := 5, [104].Area := 1, [105].Next := 116, [105].Type := 6, [105].Setup := 80, [105].Syst := 5, [105].Area := 1, [110].Type := 8, [110].Syst := 2, [110].Area := 1, [111].Next := 119, [111].Type := 6, [111].Setup := 114, [111].Syst := 2, [111].Area := 1, [112].Type := 8, [112].Syst := 3, [112].Area := 1, [113].Next := 118, [113].Type := 6, [113].Setup := 114, [113].Syst := 3, [113].Area := 1, [114].Type := 8, [114].Syst := 4, [114].Area := 1, [115].Next := 119, [115].Type := 6, [115].Setup := 114, [115].Syst := 4, [115].Area := 1, [116].Type := 8, [116].Syst := 5,
        [116].Area := 1, [117].Next := 119, [117].Type := 6, [117].Setup := 114, [117].Syst := 5, [117].Area := 1, [118].Next := 129, [118].Type := 6, [118].Setup := 82, [118].Syst := 6, [118].Area := 1, [119].Next := 129, [119].Type := 6, [119].Setup := 82, [119].Syst := 6, [119].Area := 1, [120].Type := 8, [120].Syst := 6, [120].Area := 1, [121].Next := 129, [121].Type := 6, [121].Setup := 80, [121].Syst := 6, [121].Area := 1, [122].Area := 1, [123].Next := 121, [123].Type := 1, [123].Setup := 114, [123].Syst := 6, [123].Area := 1, [123].Indx[0] := 32, [123].Indx[1] := 6, [123].Indx[2] := 32, [129].Type := 8, [129].Syst := 6, [129].Area := 1, [130].Next := 129, [130].Type := 1, [130].Setup := 64, [130].Syst := 6, [130].Area := 1, [131].Next := 132, [131].Type := 6, [131].Setup := 98, [131].Syst := 6, [131].Area := 1, [132].Type := 8, [132].Syst := 6, [132].Area := 1, [133].Next := 134, [133].Type := 1, [133].Setup := 96, [133].Syst := 7, [133].Area := 1, [134].Next := 137, [134].Type := 1, [134].Setup := 64, [134].Syst := 7, [134].Area := 1, [135].Type := 1,
        [135].Syst := 7, [135].Area := 1, [136].Type := 1, [136].Syst := 7, [136].Area := 1, [137].Next := 171, [137].Type := 1, [137].Setup := 64, [137].Syst := 7, [137].Area := 1, [138].Type := 3, [138].Syst := 7, [138].Area := 1, [140].Type := 8, [140].Syst := 7, [140].Area := 1, [141].Next := 152, [141].Type := 6, [141].Setup := 96, [141].Syst := 7, [141].Area := 1, [150].Type := 8, [150].Syst := 7, [150].Area := 1, [151].Next := 152, [151].Type := 6, [151].Setup := 96, [151].Syst := 7, [151].Area := 1, [152].Type := 8, [152].Syst := 7, [152].Area := 1, [153].Next := 20, [153].Type := 6, [153].Setup := 608, [153].Syst := 2, [153].Area := 1, [154].Next := 21, [154].Type := 6, [154].Setup := 608, [154].Syst := 2, [154].Area := 1, [155].Next := 22, [155].Type := 6, [155].Setup := 608, [155].Syst := 2, [155].Area := 1, [156].Next := 23, [156].Type := 6, [156].Setup := 608, [156].Syst := 2, [156].Area := 1, [157].Next := 24, [157].Type := 6, [157].Setup := 608, [157].Syst := 2, [157].Area := 1, [158].Next := 25, [158].Type := 6, [158].Setup := 608,
        [158].Syst := 2, [158].Area := 1, [159].Next := 26, [159].Type := 6, [159].Setup := 608, [159].Syst := 2, [159].Area := 1, [160].Next := 27, [160].Type := 6, [160].Setup := 608, [160].Syst := 2, [160].Area := 1, [161].Next := 28, [161].Type := 6, [161].Setup := 608, [161].Syst := 3, [161].Area := 1, [162].Next := 29, [162].Type := 6, [162].Setup := 608, [162].Syst := 3, [162].Area := 1, [163].Next := 30, [163].Type := 6, [163].Setup := 608, [163].Syst := 3, [163].Area := 1, [164].Next := 31, [164].Type := 6, [164].Setup := 608, [164].Syst := 3, [164].Area := 1, [165].Next := 32, [165].Type := 6, [165].Setup := 608, [165].Syst := 3, [165].Area := 1, [166].Next := 33, [166].Type := 6, [166].Setup := 608, [166].Syst := 3, [166].Area := 1, [167].Next := 34, [167].Type := 6, [167].Setup := 608, [167].Syst := 3, [167].Area := 1, [168].Next := 35, [168].Type := 6, [168].Setup := 608, [168].Syst := 3, [168].Area := 1, [170].Type := 30, [170].Setup := 64, [170].Syst := 1, [170].Area := 1, [171].Type := 30, [171].Setup := 64, [171].Syst := 1, [171].Area := 1);   // Process Flow Typologie
   automat : DINT[100] := ([0] := 40, [3] := 1835008);
        [1].0   // Partida Transporte Neumático
        [1].1   // Parada Transporte Neumático
        [2].3   // Parada Ruta Finos L6
        [2].2   // Partida Ruta Finos L6
        [2].0   // Partida Ruta Finos L5
        [2].1   // Parada Ruta Finos L5
        [0]   // CMD Selectores
   Batch : batch[10];
        [2].HEAD.DINT[5]   // Bit de linea de pelletizado
        [2].HEAD.DINT[8]   // Bit de Molienda
        [4]   // Batch Mixer
        [3]   // Batch Tolvas Harinas
        [5]   // Batch en Transporte
        [6]   // Batch en Despacho (interfaz)
   Batch_buff : batch := (Head.folio := 31, Head.orden := -3, Head.formula := 'DUMMY$00$00$00$00$00', Head.estado := 5, Head.correlativo := 1, Head.total_batch := 20, Head.peso_teorico := 1733.0, Data.codigo[0] := 81, Data.codigo[1] := 51, Data.codigo[2] := 53, Data.codigo[3] := 55, Data.codigo[4] := 57, Data.codigo[5] := 67, Data.codigo[6] := 68, Data.codigo[7] := 69, Data.codigo[8] := 70, Data.codigo[9] := 74, Data.codigo[10] := 75, Data.codigo[11] := 76, Data.codigo[12] := 77, Data.codigo[13] := 60, Data.codigo[14] := 62, Data.codigo[15] := 64, Data.codigo[16] := 66, Data.peso_f[0] := 70.0, Data.peso_f[1] := 400.0, Data.peso_f[2] := 350.0, Data.peso_f[3] := 175.0, Data.peso_f[4] := 225.0, Data.peso_f[5] := 30.0, Data.peso_f[6] := 25.0, Data.peso_f[7] := 17.5, Data.peso_f[8] := 17.5, Data.peso_f[9] := 30.0, Data.peso_f[10] := 5.0, Data.peso_f[11] := 4.0, Data.peso_f[12] := 4.0, Data.peso_f[13] := 125.0, Data.peso_f[14] := 125.0, Data.peso_f[15] := 65.0, Data.peso_f[16] := 65.0, Data.tolva[0] := 38, Data.tolva[2] := 4, Data.tolva[3] := 10, Data.tolva[4] := 12, Data.tolva[5] := 18, Data.tolva[6] := 19, Data.tolva[7] := 20, Data.tolva[8] := 21, Data.tolva[9] := 26, Data.tolva[10] := 27, Data.tolva[11] := 28, Data.tolva[12] := 29, Data.tolva[13] := 7, Data.tolva[14] := 9, Data.tolva[15] := 15, Data.tolva[16] := 17, Data.lugar[0] := 6, Data.lugar[2] := 1, Data.lugar[3] := 1,
        Data.lugar[4] := 1, Data.lugar[5] := 3, Data.lugar[6] := 3, Data.lugar[7] := 3, Data.lugar[8] := 3, Data.lugar[9] := 4, Data.lugar[10] := 4, Data.lugar[11] := 4, Data.lugar[12] := 4, Data.lugar[13] := 2, Data.lugar[14] := 2, Data.lugar[15] := 2, Data.lugar[16] := 2, Data.flags[0] := 4, Data.flags[2] := 4, Data.flags[3] := 4, Data.flags[4] := 4, Data.flags[5] := 4, Data.flags[6] := 4, Data.flags[7] := 4, Data.flags[8] := 4, Data.flags[9] := 4, Data.flags[10] := 4, Data.flags[11] := 4, Data.flags[12] := 4, Data.flags[13] := 4, Data.flags[14] := 4, Data.flags[15] := 4, Data.flags[16] := 4);
   Batch_Reportes : batch[100] := ([0].Head.folio := 12, [0].Head.orden := -2, [0].Head.formula := 'DUMMY$00$00$00$00$00', [0].Head.correlativo := 2, [0].Head.total_batch := 10, [0].Head.peso_teorico := 1201.0, [0].Data.codigo[0] := 5, [0].Data.codigo[1] := 6, [0].Data.codigo[2] := 7, [0].Data.codigo[3] := 8, [0].Data.codigo[4] := 10, [0].Data.codigo[5] := 20, [0].Data.codigo[6] := 25, [0].Data.codigo[7] := 49, [0].Data.codigo[8] := 50, [0].Data.peso_f[0] := 8.0, [0].Data.peso_f[1] := 7.0, [0].Data.peso_f[2] := 6.0, [0].Data.peso_f[3] := 5.0, [0].Data.peso_f[4] := 600.0, [0].Data.peso_f[5] := 400.0, [0].Data.peso_f[6] := 95.0, [0].Data.peso_f[7] := 30.0, [0].Data.peso_f[8] := 50.0, [0].Data.peso_r[0] := 8.085258, [0].Data.peso_r[1] := 7.1829176, [0].Data.peso_r[2] := 6.08955, [0].Data.peso_r[3] := 5.0846786, [0].Data.peso_r[4] := 601.3293, [0].Data.peso_r[5] := 408.73267, [0].Data.peso_r[6] := 6815.86, [0].Data.peso_r[7] := 30.013237, [0].Data.peso_r[8] := 50.19487, [0].Data.tolva[0] := 20, [0].Data.tolva[1] := 21, [0].Data.tolva[2] := 28, [0].Data.tolva[3] := 29, [0].Data.tolva[4] := 2, [0].Data.tolva[5] := 10, [0].Data.tolva[6] := 38, [0].Data.tolva[7] := 14, [0].Data.tolva[8] := 6, [0].Data.lugar[0] := 3, [0].Data.lugar[1] := 3, [0].Data.lugar[2] := 4, [0].Data.lugar[3] := 4, [0].Data.lugar[4] := 1, [0].Data.lugar[5] := 1, [0].Data.lugar[6] := 6, [0].Data.lugar[7] := 2, [0].Data.lugar[8] := 2, [0].Data.flags[0] := 5, [0].Data.flags[1] := 5, [0].Data.flags[2] := 5, [0].Data.flags[3] := 5, [0].Data.flags[4] := 5, [0].Data.flags[5] := 5, [0].Data.flags[6] := 5, [0].Data.flags[7] := 5, [0].Data.flags[8] := 5,
        [0].Data.fecha_i[0] := 20140321, [0].Data.fecha_i[1] := 20140321, [0].Data.fecha_i[2] := 20140321, [0].Data.fecha_i[3] := 20140321, [0].Data.fecha_i[4] := 20140321, [0].Data.fecha_i[5] := 20140321, [0].Data.fecha_i[6] := 20140321, [0].Data.fecha_i[7] := 20140321, [0].Data.fecha_i[8] := 20140321, [0].Data.fecha_f[0] := 20140321, [0].Data.fecha_f[1] := 20140321, [0].Data.fecha_f[2] := 20140321, [0].Data.fecha_f[3] := 20140321, [0].Data.fecha_f[4] := 20140321, [0].Data.fecha_f[5] := 20140321, [0].Data.fecha_f[6] := 20140321, [0].Data.fecha_f[7] := 20140321, [0].Data.fecha_f[8] := 20140321, [0].Data.hora_i[0] := 12443466, [0].Data.hora_i[1] := 13125216, [0].Data.hora_i[2] := 12443466, [0].Data.hora_i[3] := 13122756, [0].Data.hora_i[4] := 12443466, [0].Data.hora_i[5] := 13125706, [0].Data.hora_i[6] := 13334183, [0].Data.hora_i[7] := 12443466, [0].Data.hora_i[8] := 13125486, [0].Data.hora_f[0] := 12450236, [0].Data.hora_f[1] := 13215516, [0].Data.hora_f[2] := 12450006, [0].Data.hora_f[3] := 13214826, [0].Data.hora_f[4] := 13121366, [0].Data.hora_f[5] := 13131736, [0].Data.hora_f[6] := 14305313, [0].Data.hora_f[7] := 12450406, [0].Data.hora_f[8] := 13130766, [1].Head.folio := 13, [1].Head.orden := -2, [1].Head.formula := 'DUMMY$00$00$00$00$00', [1].Head.correlativo := 3, [1].Head.total_batch := 10, [1].Head.peso_teorico := 1201.0, [1].Data.codigo[0] := 5, [1].Data.codigo[1] := 6, [1].Data.codigo[2] := 7, [1].Data.codigo[3] := 8, [1].Data.codigo[4] := 10, [1].Data.codigo[5] := 20, [1].Data.codigo[6] := 25, [1].Data.codigo[7] := 49, [1].Data.codigo[8] := 50, [1].Data.peso_f[0] := 8.0, [1].Data.peso_f[1] := 7.0, [1].Data.peso_f[2] := 6.0, [1].Data.peso_f[3] := 5.0, [1].Data.peso_f[4] := 600.0, [1].Data.peso_f[5] := 400.0, [1].Data.peso_f[6] := 95.0, [1].Data.peso_f[7] := 30.0, [1].Data.peso_f[8] := 50.0,
        [1].Data.peso_r[1] := 6.981835, [1].Data.peso_r[2] := 6.088384, [1].Data.peso_r[3] := 5.0858264, [1].Data.peso_r[4] := 606.447, [1].Data.peso_r[5] := 413.8863, [1].Data.peso_r[6] := 95.70117, [1].Data.peso_r[7] := 30.00908, [1].Data.peso_r[8] := 50.574806, [1].Data.tolva[1] := 21, [1].Data.tolva[2] := 28, [1].Data.tolva[3] := 29, [1].Data.tolva[4] := 2, [1].Data.tolva[5] := 10, [1].Data.tolva[6] := 38, [1].Data.tolva[7] := 14, [1].Data.tolva[8] := 6, [1].Data.lugar[1] := 3, [1].Data.lugar[2] := 4, [1].Data.lugar[3] := 4, [1].Data.lugar[4] := 1, [1].Data.lugar[5] := 1, [1].Data.lugar[6] := 6, [1].Data.lugar[7] := 2, [1].Data.lugar[8] := 2, [1].Data.flags[0] := 2, [1].Data.flags[1] := 5, [1].Data.flags[2] := 5, [1].Data.flags[3] := 5, [1].Data.flags[4] := 21, [1].Data.flags[5] := 5, [1].Data.flags[6] := 5, [1].Data.flags[7] := 5, [1].Data.flags[8] := 5, [1].Data.fecha_i[0] := 20140321, [1].Data.fecha_i[1] := 20140321, [1].Data.fecha_i[2] := 20140321, [1].Data.fecha_i[3] := 20140321, [1].Data.fecha_i[4] := 20140321, [1].Data.fecha_i[5] := 20140324, [1].Data.fecha_i[6] := 20140324, [1].Data.fecha_i[7] := 20140321, [1].Data.fecha_i[8] := 20140324, [1].Data.fecha_f[1] := 20140321, [1].Data.fecha_f[2] := 20140321, [1].Data.fecha_f[3] := 20140321, [1].Data.fecha_f[4] := 20140321, [1].Data.fecha_f[5] := 20140324, [1].Data.fecha_f[6] := 20140324, [1].Data.fecha_f[7] := 20140321, [1].Data.fecha_f[8] := 20140324, [1].Data.hora_i[0] := 13261586, [1].Data.hora_i[1] := 18003263, [1].Data.hora_i[2] := 18003263, [1].Data.hora_i[3] := 18004183, [1].Data.hora_i[4] := 18003263, [1].Data.hora_i[5] := 10441523, [1].Data.hora_i[6] := 10453303, [1].Data.hora_i[7] := 18003263, [1].Data.hora_i[8] := 10435383, [1].Data.hora_f[1] := 18004523,
        [1].Data.hora_f[2] := 18004053, [1].Data.hora_f[3] := 18005273, [1].Data.hora_f[4] := 18005143, [1].Data.hora_f[5] := 10443303, [1].Data.hora_f[6] := 10472743, [1].Data.hora_f[7] := 18004153, [1].Data.hora_f[8] := 10441493, [2].Head.folio := 14, [2].Head.orden := -2, [2].Head.formula := 'DUMMY$00$00$00$00$00', [2].Head.correlativo := 4, [2].Head.total_batch := 10, [2].Head.peso_teorico := 1201.0, [2].Data.codigo[0] := 5, [2].Data.codigo[1] := 6, [2].Data.codigo[2] := 7, [2].Data.codigo[3] := 8, [2].Data.codigo[4] := 10, [2].Data.codigo[5] := 20, [2].Data.codigo[6] := 25, [2].Data.codigo[7] := 49, [2].Data.codigo[8] := 50, [2].Data.peso_f[0] := 8.0, [2].Data.peso_f[1] := 7.0, [2].Data.peso_f[2] := 6.0, [2].Data.peso_f[3] := 5.0, [2].Data.peso_f[4] := 600.0, [2].Data.peso_f[5] := 400.0, [2].Data.peso_f[6] := 95.0, [2].Data.peso_f[7] := 30.0, [2].Data.peso_f[8] := 50.0, [2].Data.peso_r[0] := 7.9872093, [2].Data.peso_r[1] := 6.981963, [2].Data.peso_r[2] := 6.0895605, [2].Data.peso_r[3] := 4.979808, [2].Data.peso_r[4] := 606.04663, [2].Data.peso_r[5] := 409.1341, [2].Data.peso_r[6] := 95.691895, [2].Data.peso_r[7] := 30.018162, [2].Data.peso_r[8] := 50.19932, [2].Data.tolva[0] := 20, [2].Data.tolva[1] := 21, [2].Data.tolva[2] := 28, [2].Data.tolva[3] := 29, [2].Data.tolva[4] := 2, [2].Data.tolva[5] := 10, [2].Data.tolva[6] := 38, [2].Data.tolva[7] := 14, [2].Data.tolva[8] := 6, [2].Data.lugar[0] := 3, [2].Data.lugar[1] := 3, [2].Data.lugar[2] := 4, [2].Data.lugar[3] := 4, [2].Data.lugar[4] := 1, [2].Data.lugar[5] := 1, [2].Data.lugar[6] := 6, [2].Data.lugar[7] := 2, [2].Data.lugar[8] := 2, [2].Data.flags[0] := 5, [2].Data.flags[1] := 5,
        [2].Data.flags[2] := 5, [2].Data.flags[3] := 5, [2].Data.flags[4] := 5, [2].Data.flags[5] := 5, [2].Data.flags[6] := 5, [2].Data.flags[7] := 5, [2].Data.flags[8] := 5, [2].Data.fecha_i[0] := 20140324, [2].Data.fecha_i[1] := 20140324, [2].Data.fecha_i[2] := 20140324, [2].Data.fecha_i[3] := 20140324, [2].Data.fecha_i[4] := 20140324, [2].Data.fecha_i[5] := 20140324, [2].Data.fecha_i[6] := 20140324, [2].Data.fecha_i[7] := 20140324, [2].Data.fecha_i[8] := 20140324, [2].Data.fecha_f[0] := 20140324, [2].Data.fecha_f[1] := 20140324, [2].Data.fecha_f[2] := 20140324, [2].Data.fecha_f[3] := 20140324, [2].Data.fecha_f[4] := 20140324, [2].Data.fecha_f[5] := 20140324, [2].Data.fecha_f[6] := 20140324, [2].Data.fecha_f[7] := 20140324, [2].Data.fecha_f[8] := 20140324, [2].Data.hora_i[0] := 10515543, [2].Data.hora_i[1] := 10520533, [2].Data.hora_i[2] := 10515543, [2].Data.hora_i[3] := 10520373, [2].Data.hora_i[4] := 10515543, [2].Data.hora_i[5] := 10521563, [2].Data.hora_i[6] := 10533033, [2].Data.hora_i[7] := 10515543, [2].Data.hora_i[8] := 10520473, [2].Data.hora_f[0] := 10520493, [2].Data.hora_f[1] := 10521793, [2].Data.hora_f[2] := 10520333, [2].Data.hora_f[3] := 10521483, [2].Data.hora_f[4] := 10521523, [2].Data.hora_f[5] := 10522963, [2].Data.hora_f[6] := 10550063, [2].Data.hora_f[7] := 10520433, [2].Data.hora_f[8] := 10521743, [3].Head.folio := 15, [3].Head.orden := -2, [3].Head.formula := 'DUMMY$00$00$00$00$00', [3].Head.correlativo := 5, [3].Head.total_batch := 10, [3].Head.peso_teorico := 1201.0, [3].Data.codigo[0] := 5, [3].Data.codigo[1] := 6, [3].Data.codigo[2] := 7, [3].Data.codigo[3] := 8, [3].Data.codigo[4] := 10, [3].Data.codigo[5] := 20, [3].Data.codigo[6] := 25, [3].Data.codigo[7] := 49, [3].Data.codigo[8] := 50, [3].Data.peso_f[0] := 8.0, [3].Data.peso_f[1] := 7.0,
        [3].Data.peso_f[2] := 6.0, [3].Data.peso_f[3] := 5.0, [3].Data.peso_f[4] := 600.0, [3].Data.peso_f[5] := 400.0, [3].Data.peso_f[6] := 95.0, [3].Data.peso_f[7] := 30.0, [3].Data.peso_f[8] := 50.0, [3].Data.peso_r[0] := 7.9849377, [3].Data.peso_r[1] := 6.9808035, [3].Data.peso_r[2] := 6.088262, [3].Data.peso_r[3] := 4.979818, [3].Data.peso_r[4] := 606.44684, [3].Data.peso_r[5] := 408.625, [3].Data.peso_r[6] := 95.495605, [3].Data.peso_r[7] := 30.013268, [3].Data.peso_r[8] := 50.195526, [3].Data.tolva[0] := 20, [3].Data.tolva[1] := 21, [3].Data.tolva[2] := 28, [3].Data.tolva[3] := 29, [3].Data.tolva[4] := 2, [3].Data.tolva[5] := 10, [3].Data.tolva[6] := 38, [3].Data.tolva[7] := 14, [3].Data.tolva[8] := 6, [3].Data.lugar[0] := 3, [3].Data.lugar[1] := 3, [3].Data.lugar[2] := 4, [3].Data.lugar[3] := 4, [3].Data.lugar[4] := 1, [3].Data.lugar[5] := 1, [3].Data.lugar[6] := 6, [3].Data.lugar[7] := 2, [3].Data.lugar[8] := 2, [3].Data.flags[0] := 5, [3].Data.flags[1] := 5, [3].Data.flags[2] := 5, [3].Data.flags[3] := 5, [3].Data.flags[4] := 5, [3].Data.flags[5] := 5, [3].Data.flags[6] := 5, [3].Data.flags[7] := 5, [3].Data.flags[8] := 5, [3].Data.fecha_i[0] := 20140324, [3].Data.fecha_i[1] := 20140324, [3].Data.fecha_i[2] := 20140324, [3].Data.fecha_i[3] := 20140324, [3].Data.fecha_i[4] := 20140324, [3].Data.fecha_i[5] := 20140324, [3].Data.fecha_i[6] := 20140324, [3].Data.fecha_i[7] := 20140324, [3].Data.fecha_i[8] := 20140324, [3].Data.fecha_f[0] := 20140324, [3].Data.fecha_f[1] := 20140324, [3].Data.fecha_f[2] := 20140324, [3].Data.fecha_f[3] := 20140324, [3].Data.fecha_f[4] := 20140324, [3].Data.fecha_f[5] := 20140324, [3].Data.fecha_f[6] := 20140324, [3].Data.fecha_f[7] := 20140324,
        [3].Data.fecha_f[8] := 20140324, [3].Data.hora_i[0] := 10564023, [3].Data.hora_i[1] := 10565003, [3].Data.hora_i[2] := 10564023, [3].Data.hora_i[3] := 10564843, [3].Data.hora_i[4] := 10564023, [3].Data.hora_i[5] := 10565663, [3].Data.hora_i[6] := 10581953, [3].Data.hora_i[7] := 10564023, [3].Data.hora_i[8] := 10564943, [3].Data.hora_f[0] := 10564963, [3].Data.hora_f[1] := 10570233, [3].Data.hora_f[2] := 10564803, [3].Data.hora_f[3] := 10565953, [3].Data.hora_f[4] := 10565623, [3].Data.hora_f[5] := 10571923, [3].Data.hora_f[6] := 10592963, [3].Data.hora_f[7] := 10564903, [3].Data.hora_f[8] := 10570213, [4].Head.folio := 16, [4].Head.orden := -2, [4].Head.formula := 'DUMMY$00$00$00$00$00', [4].Head.correlativo := 6, [4].Head.total_batch := 10, [4].Head.peso_teorico := 1201.0, [4].Data.codigo[0] := 5, [4].Data.codigo[1] := 6, [4].Data.codigo[2] := 7, [4].Data.codigo[3] := 8, [4].Data.codigo[4] := 10, [4].Data.codigo[5] := 20, [4].Data.codigo[6] := 25, [4].Data.codigo[7] := 49, [4].Data.codigo[8] := 50, [4].Data.peso_f[0] := 8.0, [4].Data.peso_f[1] := 7.0, [4].Data.peso_f[2] := 6.0, [4].Data.peso_f[3] := 5.0, [4].Data.peso_f[4] := 600.0, [4].Data.peso_f[5] := 400.0, [4].Data.peso_f[6] := 95.0, [4].Data.peso_f[7] := 30.0, [4].Data.peso_f[8] := 50.0, [4].Data.peso_r[0] := 8.085273, [4].Data.peso_r[1] := 7.18291, [4].Data.peso_r[2] := 5.9840455, [4].Data.peso_r[3] := 5.084679, [4].Data.peso_r[4] := 606.2944, [4].Data.peso_r[5] := 408.6775, [4].Data.peso_r[6] := 95.60205, [4].Data.peso_r[7] := 30.417713, [4].Data.peso_r[8] := 50.199627, [4].Data.tolva[0] := 20, [4].Data.tolva[1] := 21, [4].Data.tolva[2] := 28, [4].Data.tolva[3] := 29, [4].Data.tolva[4] := 2, [4].Data.tolva[5] := 10, [4].Data.tolva[6] := 38, [4].Data.tolva[7] := 14,
        [4].Data.tolva[8] := 6, [4].Data.lugar[0] := 3, [4].Data.lugar[1] := 3, [4].Data.lugar[2] := 4, [4].Data.lugar[3] := 4, [4].Data.lugar[4] := 1, [4].Data.lugar[5] := 1, [4].Data.lugar[6] := 6, [4].Data.lugar[7] := 2, [4].Data.lugar[8] := 2, [4].Data.flags[0] := 5, [4].Data.flags[1] := 5, [4].Data.flags[2] := 5, [4].Data.flags[3] := 5, [4].Data.flags[4] := 5, [4].Data.flags[5] := 5, [4].Data.flags[6] := 5, [4].Data.flags[7] := 5, [4].Data.flags[8] := 5, [4].Data.fecha_i[0] := 20140324, [4].Data.fecha_i[1] := 20140324, [4].Data.fecha_i[2] := 20140324, [4].Data.fecha_i[3] := 20140324, [4].Data.fecha_i[4] := 20140324, [4].Data.fecha_i[5] := 20140324, [4].Data.fecha_i[6] := 20140324, [4].Data.fecha_i[7] := 20140324, [4].Data.fecha_i[8] := 20140324, [4].Data.fecha_f[0] := 20140324, [4].Data.fecha_f[1] := 20140324, [4].Data.fecha_f[2] := 20140324, [4].Data.fecha_f[3] := 20140324, [4].Data.fecha_f[4] := 20140324, [4].Data.fecha_f[5] := 20140324, [4].Data.fecha_f[6] := 20140324, [4].Data.fecha_f[7] := 20140324, [4].Data.fecha_f[8] := 20140324, [4].Data.hora_i[0] := 10581963, [4].Data.hora_i[1] := 10582943, [4].Data.hora_i[2] := 10581963, [4].Data.hora_i[3] := 10582773, [4].Data.hora_i[4] := 10581963, [4].Data.hora_i[5] := 10583983, [4].Data.hora_i[6] := 11010393, [4].Data.hora_i[7] := 10581963, [4].Data.hora_i[8] := 10582883, [4].Data.hora_f[0] := 10582903, [4].Data.hora_f[1] := 10584723, [4].Data.hora_f[2] := 10582733, [4].Data.hora_f[3] := 10583893, [4].Data.hora_f[4] := 10583943, [4].Data.hora_f[5] := 10585743, [4].Data.hora_f[6] := 11024303, [4].Data.hora_f[7] := 10582843, [4].Data.hora_f[8] := 10584143, [5].Head.folio := 17, [5].Head.orden := -2, [5].Head.formula := 'DUMMY$00$00$00$00$00', [5].Head.correlativo := 7, [5].Head.total_batch := 10,
        [5].Head.peso_teorico := 1201.0, [5].Data.codigo[0] := 5, [5].Data.codigo[1] := 6, [5].Data.codigo[2] := 7, [5].Data.codigo[3] := 8, [5].Data.codigo[4] := 10, [5].Data.codigo[5] := 20, [5].Data.codigo[6] := 25, [5].Data.codigo[7] := 49, [5].Data.codigo[8] := 50, [5].Data.peso_f[0] := 8.0, [5].Data.peso_f[1] := 7.0, [5].Data.peso_f[2] := 6.0, [5].Data.peso_f[3] := 5.0, [5].Data.peso_f[4] := 600.0, [5].Data.peso_f[5] := 400.0, [5].Data.peso_f[6] := 95.0, [5].Data.peso_f[7] := 30.0, [5].Data.peso_f[8] := 50.0, [5].Data.peso_r[0] := 8.08628, [5].Data.peso_r[1] := 6.980831, [5].Data.peso_r[2] := 5.983946, [5].Data.peso_r[3] := 4.9797, [5].Data.peso_r[4] := 601.3783, [5].Data.peso_r[5] := 404.00012, [5].Data.peso_r[6] := 95.60603, [5].Data.peso_r[7] := 30.421803, [5].Data.peso_r[8] := 50.19488, [5].Data.tolva[0] := 20, [5].Data.tolva[1] := 21, [5].Data.tolva[2] := 28, [5].Data.tolva[3] := 29, [5].Data.tolva[4] := 2, [5].Data.tolva[5] := 10, [5].Data.tolva[6] := 38, [5].Data.tolva[7] := 14, [5].Data.tolva[8] := 6, [5].Data.lugar[0] := 3, [5].Data.lugar[1] := 3, [5].Data.lugar[2] := 4, [5].Data.lugar[3] := 4, [5].Data.lugar[4] := 1, [5].Data.lugar[5] := 1, [5].Data.lugar[6] := 6, [5].Data.lugar[7] := 2, [5].Data.lugar[8] := 2, [5].Data.flags[0] := 5, [5].Data.flags[1] := 5, [5].Data.flags[2] := 5, [5].Data.flags[3] := 5, [5].Data.flags[4] := 5, [5].Data.flags[5] := 5, [5].Data.flags[6] := 5, [5].Data.flags[7] := 5, [5].Data.flags[8] := 5, [5].Data.fecha_i[0] := 20140324, [5].Data.fecha_i[1] := 20140324, [5].Data.fecha_i[2] := 20140324, [5].Data.fecha_i[3] := 20140324, [5].Data.fecha_i[4] := 20140324,
        [5].Data.fecha_i[5] := 20140324, [5].Data.fecha_i[6] := 20140324, [5].Data.fecha_i[7] := 20140324, [5].Data.fecha_i[8] := 20140324, [5].Data.fecha_f[0] := 20140324, [5].Data.fecha_f[1] := 20140324, [5].Data.fecha_f[2] := 20140324, [5].Data.fecha_f[3] := 20140324, [5].Data.fecha_f[4] := 20140324, [5].Data.fecha_f[5] := 20140324, [5].Data.fecha_f[6] := 20140324, [5].Data.fecha_f[7] := 20140324, [5].Data.fecha_f[8] := 20140324, [5].Data.hora_i[0] := 11010403, [5].Data.hora_i[1] := 11011383, [5].Data.hora_i[2] := 11010403, [5].Data.hora_i[3] := 11011213, [5].Data.hora_i[4] := 11010403, [5].Data.hora_i[5] := 11013163, [5].Data.hora_i[6] := 11042193, [5].Data.hora_i[7] := 11010403, [5].Data.hora_i[8] := 11011323, [5].Data.hora_f[0] := 11011343, [5].Data.hora_f[1] := 11012633, [5].Data.hora_f[2] := 11011173, [5].Data.hora_f[3] := 11012323, [5].Data.hora_f[4] := 11013123, [5].Data.hora_f[5] := 11014503, [5].Data.hora_f[6] := 11054733, [5].Data.hora_f[7] := 11011283, [5].Data.hora_f[8] := 11012583, [6].Head.folio := 18, [6].Head.orden := -2, [6].Head.formula := 'DUMMY$00$00$00$00$00', [6].Head.correlativo := 8, [6].Head.total_batch := 10, [6].Head.peso_teorico := 1201.0, [6].Data.codigo[0] := 5, [6].Data.codigo[1] := 6, [6].Data.codigo[2] := 7, [6].Data.codigo[3] := 8, [6].Data.codigo[4] := 10, [6].Data.codigo[5] := 20, [6].Data.codigo[6] := 25, [6].Data.codigo[7] := 49, [6].Data.codigo[8] := 50, [6].Data.peso_f[0] := 8.0, [6].Data.peso_f[1] := 7.0, [6].Data.peso_f[2] := 6.0, [6].Data.peso_f[3] := 5.0, [6].Data.peso_f[4] := 600.0, [6].Data.peso_f[5] := 400.0, [6].Data.peso_f[6] := 95.0, [6].Data.peso_f[7] := 30.0, [6].Data.peso_f[8] := 50.0, [6].Data.peso_r[0] := 8.087415, [6].Data.peso_r[1] := 6.9818544, [6].Data.peso_r[2] := 5.985111, [6].Data.peso_r[3] := 4.980858, [6].Data.peso_r[4] := 601.4355,
        [6].Data.peso_r[5] := 403.89203, [6].Data.peso_r[6] := 94.60004, [6].Data.peso_r[7] := 30.422052, [6].Data.peso_r[8] := 50.19529, [6].Data.tolva[0] := 20, [6].Data.tolva[1] := 21, [6].Data.tolva[2] := 28, [6].Data.tolva[3] := 29, [6].Data.tolva[4] := 2, [6].Data.tolva[5] := 10, [6].Data.tolva[6] := 38, [6].Data.tolva[7] := 14, [6].Data.tolva[8] := 6, [6].Data.lugar[0] := 3, [6].Data.lugar[1] := 3, [6].Data.lugar[2] := 4, [6].Data.lugar[3] := 4, [6].Data.lugar[4] := 1, [6].Data.lugar[5] := 1, [6].Data.lugar[6] := 6, [6].Data.lugar[7] := 2, [6].Data.lugar[8] := 2, [6].Data.flags[0] := 5, [6].Data.flags[1] := 5, [6].Data.flags[2] := 5, [6].Data.flags[3] := 5, [6].Data.flags[4] := 5, [6].Data.flags[5] := 5, [6].Data.flags[6] := 5, [6].Data.flags[7] := 5, [6].Data.flags[8] := 5, [6].Data.fecha_i[0] := 20140324, [6].Data.fecha_i[1] := 20140324, [6].Data.fecha_i[2] := 20140324, [6].Data.fecha_i[3] := 20140324, [6].Data.fecha_i[4] := 20140324, [6].Data.fecha_i[5] := 20140324, [6].Data.fecha_i[6] := 20140324, [6].Data.fecha_i[7] := 20140324, [6].Data.fecha_i[8] := 20140324, [6].Data.fecha_f[0] := 20140324, [6].Data.fecha_f[1] := 20140324, [6].Data.fecha_f[2] := 20140324, [6].Data.fecha_f[3] := 20140324, [6].Data.fecha_f[4] := 20140324, [6].Data.fecha_f[5] := 20140324, [6].Data.fecha_f[6] := 20140324, [6].Data.fecha_f[7] := 20140324, [6].Data.fecha_f[8] := 20140324, [6].Data.hora_i[0] := 11042203, [6].Data.hora_i[1] := 11043183, [6].Data.hora_i[2] := 11042203, [6].Data.hora_i[3] := 11043023, [6].Data.hora_i[4] := 11042203, [6].Data.hora_i[5] := 11044153, [6].Data.hora_i[6] := 11072673, [6].Data.hora_i[7] := 11042203, [6].Data.hora_i[8] := 11043123, [6].Data.hora_f[0] := 11043143, [6].Data.hora_f[1] := 11044433,
        [6].Data.hora_f[2] := 11042983, [6].Data.hora_f[3] := 11044123, [6].Data.hora_f[4] := 11044113, [6].Data.hora_f[5] := 11045543, [6].Data.hora_f[6] := 11082133, [6].Data.hora_f[7] := 11043083, [6].Data.hora_f[8] := 11044383, [7].Head.folio := 19, [7].Head.orden := -2, [7].Head.formula := 'DUMMY$00$00$00$00$00', [7].Head.correlativo := 9, [7].Head.total_batch := 10, [7].Head.peso_teorico := 1201.0, [7].Data.codigo[0] := 5, [7].Data.codigo[1] := 6, [7].Data.codigo[2] := 7, [7].Data.codigo[3] := 8, [7].Data.codigo[4] := 10, [7].Data.codigo[5] := 20, [7].Data.codigo[6] := 25, [7].Data.codigo[7] := 49, [7].Data.codigo[8] := 50, [7].Data.peso_f[0] := 8.0, [7].Data.peso_f[1] := 7.0, [7].Data.peso_f[2] := 6.0, [7].Data.peso_f[3] := 5.0, [7].Data.peso_f[4] := 600.0, [7].Data.peso_f[5] := 400.0, [7].Data.peso_f[6] := 95.0, [7].Data.peso_f[7] := 30.0, [7].Data.peso_f[8] := 50.0, [7].Data.peso_r[0] := 8.087537, [7].Data.peso_r[1] := 6.981844, [7].Data.peso_r[2] := 5.9851527, [7].Data.peso_r[3] := 5.084555, [7].Data.peso_r[4] := 601.33405, [7].Data.peso_r[5] := 403.9477, [7].Data.peso_r[6] := 94.60004, [7].Data.peso_r[7] := 29.588737, [7].Data.peso_r[8] := 50.195244, [7].Data.tolva[0] := 20, [7].Data.tolva[1] := 21, [7].Data.tolva[2] := 28, [7].Data.tolva[3] := 29, [7].Data.tolva[4] := 2, [7].Data.tolva[5] := 10, [7].Data.tolva[6] := 38, [7].Data.tolva[7] := 14, [7].Data.tolva[8] := 6, [7].Data.lugar[0] := 3, [7].Data.lugar[1] := 3, [7].Data.lugar[2] := 4, [7].Data.lugar[3] := 4, [7].Data.lugar[4] := 1, [7].Data.lugar[5] := 1, [7].Data.lugar[6] := 6, [7].Data.lugar[7] := 2, [7].Data.lugar[8] := 2, [7].Data.flags[0] := 5, [7].Data.flags[1] := 5,
